(* CODESYS project PRO_JSON 1.0.20.0 Codesys SP17.library
   DocFormat: reStructuredText
   Company: Pro Electric
   DefaultNamespace: PRO_JSON
   Placeholder: PRO_JSON
   Author: TVM
   Description: Patched by Risele
   Version: 1.0.20.0
   Title: PRO JSON

Project tree, tasks and I/O mapping:
  libraries: Standard, 3.5.18.0 (System); StringUtils, 3.5.20.0 (System); SysMem, 3.5.17.0 (System); VisuDialogs, * (System)
  Data Types/
    data type ASCII
    data type JSONNAMEVALUE
    data type JSONVALUETYPE
    function block JSONVAR [ST]: FirstLevel, VarName, ValueType, Null, Number, Boolean, Integer, CharString, UInteger, Format, ApplicationLevel, LastIndex, ProgramLevel, AsUnicode, AsHexString, AsString, AsDWord, AsDateTime, Size, TestInit, Init, IsFirstVar, CreateNamesArray, FB_Init, GetArrayIndex
    data type JSONVARINFO
    data type JSONFORMAT
    data type ARRAY_INDEX
  Examples/
    data type EXAMPLEJSONSTRUCT
    data type EXAMPLEJSONSTRUCT_1
    program ExampleJSON_PRG [ST]
    function block EXAMPLE_FB [ST]
    program Test_ArrayOfStruct_PRG [ST]
    program Test_Array_PRG [ST]
    program Test_NestedStruct_PRG [ST]
    program Test_SingleVar_PRG [ST]
    program Test_Struct_PRG [ST]
    data type ARRAYOFSTRUCT
    data type JSONSTRUCT
    data type JSONSTRUCT_1
  Functions/
    function CLEANSTRING [ST]
    function ISBOOLEAN [ST]
    function ISNUMBER [ST]
    function REAL_TO_STRING_X [ST]
    function SPLIT_VARNAME [ST]
    function ISINTEGER [ST]
    function JSONVALUE_TO_STRING [ST]
    function STRING_TO_JSONVALUE [ST]
    function MATCH_NAMES [ST]
    function HEXSTR_TO_UDINT [ST]
    function ISHEX [ST]
    function UDINT_TO_HEXSTR [ST]
    function FORMAT_JSON [ST]
    function HEX4_TO_UINT [ST]
    function UINT_TO_HEX4 [ST]
    function VALUETYPE_FROM_STRING [ST]
    function ISNULL [ST]
    function DWORD_TO_HEXSTR [ST]
    function IEC_TO_JSON [ST]
    function JSON_TO_IEC [ST]
    function DWORD_TO_UNICODE [ST]
    function ARRAY_INDEXES_EQUAL [ST]
    function ARRAY_INDEXES_LESS [ST]
    function CLEAR_ARRAY_INDEX_VECTOR [ST]
  global variables GPL_JSON
  program Notes [ST]
  Visualizations/
    visualisation JSON_TO_STRUCT_VISU
    visualisation STRUCT_TO_JSON_VISU
    visualisation JSONVARS_TABLE_VISU
    visualisation JSONVAR_TABLE_VISU
    text list ValueType_Textlist
  text list GlobalTextList
  Function Blocks/
    function block JSON_TO_STRUCT [ST]: ClearAll, Value, FindValueStartPosition, GetValueAsString, FindValueStopPosition, ErrorHandler, ClearNameValue, CheckApplicationName, CheckMaxVars, CheckPointers, MatchAllLevels, CloseObject, OpenArray, Comma, CloseArray, OpenObject, Name
    function block STRUCT_TO_JSON [ST]: FindMaxLevel, CreateArray, CreateObject, CreateValue, CreateName, HasNonNullDescendant, PrependComma, Initialize, InitJsonVars, CheckMaxVars, CheckApplicationName, CheckPointers, FindMatchingClose, CloseArray, CloseObject, ClearString
*)

// Data Types/ASCII
///
///| Author: Tim Van Meppelen, Pro Electric Inc.
///| timv@proelectric.com
///| Date: Nov 2, 2018
///| enumeration of all ascii characters
TYPE ASCII :
(
	NULL := 0,
	SOH := 1,
	STX := 2,
	ETX := 3,
	EOT := 4,
	ENQ := 5,
	ACK := 6,
	BEL := 7,
	BS := 8,
	HT := 9,
	LF := 10,
	VT := 11,
	FF := 12,
	CR := 13,
	SO := 14,
	SI := 15,
	DLE := 16,
	DC1 := 17,
	DC2 := 18,
	DC3 := 19,
	DC4 := 20,
	NAK := 21,
	SYN := 22,
	ETB := 23,
	CAN := 24,
	EM := 25,
	SUB_ := 26,
	ESC := 27,
	FS := 28,
	GS := 29,
	RS := 30,
	US := 31,
	SPACE := 32,
	BANG := 33,
	DOUBLE_QUOTE := 34,
	HASH := 35,
	DOLLAR := 36,
	PERCENT := 37,
	AMPERSAND := 38,
	SINGLE_QUOTE := 39,
	OPEN_PAREN := 40,
	CLOSE_PAREN := 41,
	STAR := 42,
	PLUS := 43,
	COMMA := 44,
	MINUS := 45,
	DOT := 46,
	SLASH := 47,
	_0 := 48,
	_1 := 49,
	_2 := 50,
	_3 := 51,
	_4 := 52,
	_5 := 53,
	_6 := 54,
	_7 := 55,
	_8 := 56,
	_9 := 57,
	COLON := 58,
	SEMICOLON := 59,
	LESS_THAN := 60,
	EQUALS := 61,
	GREATER_THAN := 62,
	QUESTION := 63,
	AT_SIGN := 64,
	_A := 65,
	_B := 66,
	_C := 67,
	_D := 68,
	_E := 69,
	_F := 70,
	_G := 71,
	_H := 72,
	_I := 73,
	_J := 74,
	_K := 75,
	_L := 76,
	_M := 77,
	_N := 78,
	_O := 79,
	_P := 80,
	_Q := 81,
	_R := 82,
	_S := 83,
	_T := 84,
	_U := 85,
	_V := 86,
	_W := 87,
	_X := 88,
	_Y := 89,
	_Z := 90,
	OPEN_BRACKET := 91,
	BACKSLASH := 92,
	CLOSE_BRACKET := 93,
	CARET := 94,
	UNDERSCORE := 95,
	BACKQUOTE := 96,
	_a_ := 97,
	_b_ := 98,
	_c_ := 99,
	_d_ := 100,
	_e_ := 101,
	_f_ := 102,
	_g_ := 103,
	_h_ := 104,
	_i_ := 105,
	_j_ := 106,
	_k_ := 107,
	_l_ := 108,
	_m_ := 109,
	_n_ := 110,
	_o_ := 111,
	_p_ := 112,
	_q_ := 113,
	_r_ := 114,
	_s_ := 115,
	_t_ := 116,
	_u_ := 117,
	_v_ := 118,
	_w_ := 119,
	_x_ := 120,
	_y_ := 121,
	_z_ := 122,
	OPEN_BRACE := 123,
	PIPE := 124,
	CLOSE_BRACE := 125,
	TILDE := 126,
	DEL := 127
) BYTE;
END_TYPE

// Data Types/JSONNAMEVALUE
///
///| Author: Tim Van Meppelen, Pro Electric Inc.
///| timv@proelectric.com
///| Date: Nov 2, 2018
///| name : value pair
TYPE JSONNAMEVALUE :
STRUCT
	///name of the object at this level
	Name: STRING(GPL_JSON.MAX_NAME_SIZE);
	///value of the object at this level
	Value: STRING(GPL_JSON.MAX_VALUE_SIZE);
	///array index of the object at this level
	ArrayIndex: ARRAY_INDEX := ARRAY_INDEX.Invalid;
	IsArray: BOOL;
	ArrayDimCount: UINT := 0;
	ArrayIndexes: ARRAY[1..GPL_JSON.MAX_ARRAY_DIMENSIONS] OF INT;
END_STRUCT
END_TYPE

// Data Types/JSONVALUETYPE
///
///| Author: Tim Van Meppelen, Pro Electric Inc.
///| timv@proelectric.com
///| Date: Nov 2, 2018
///| enumeration of all json types
///| NOTE: JSON standard is somewhat ambiguous with number types, so integer and floating point numbers are separate types in this library
TYPE JSONVALUETYPE :
(
	///local var is type STRING
	json_string,
	///local var is REAL
	json_number,
	///local var is DINT
	json_integer,
	///locar var is UDINT	(new type by Fabrizio Morlino)
	json_uinteger,
	///local var is BOOL
	json_boolean,
	///local var is type null
	json_null,
	///object is an array
	json_array,
	///object is another object (nested objects)
	json_object
);
END_TYPE

// Data Types/JSONVARINFO
///
///| Author: Tim Van Meppelen, Pro Electric Inc.
///| timv@proelectric.com
///| Date: Nov 2, 2018
///| variable info structure, used with JSONVAR
TYPE JSONVARINFO :
STRUCT
	///name of this variable or object
	Name: STRING(GPL_JSON.MAX_NAME_SIZE);
	///first variable of a new object
	NewObject: BOOL;
	///variable in an object
	InObject: BOOL;
	///last variable of an object
	EndObject: BOOL;
	///array index of the object at this level	
	ArrayIndex: ARRAY_INDEX := ARRAY_INDEX.Invalid;
	///first variable of a new array
	NewArray: BOOL;
	///variable in an array
	InArray: BOOL;
	///last variable of an array
	EndArray: BOOL;
	/// 0 = not in array, 1..MAX_ARRAY_DIMENSIONS otherwise
	ArrayDimCount: UINT := 0;
	/// full multidim index vector
	ArrayIndexes: ARRAY[1..GPL_JSON.MAX_ARRAY_DIMENSIONS] OF INT;
END_STRUCT
END_TYPE

// Examples/EXAMPLEJSONSTRUCT
///
///| Author: Tim Van Meppelen, Pro Electric Inc.
///| timv@proelectric.com
///| Date: Jan 31, 2020
///| example of a struct of json variables
TYPE EXAMPLEJSONSTRUCT :
STRUCT
	var1: JSONVAR;
	var2: JSONVAR;
	var3: JSONVAR;
	obj: EXAMPLEJSONSTRUCT_1;
	arrayobj: ARRAY[1..3] OF JSONVAR;
END_STRUCT
END_TYPE

// Examples/EXAMPLEJSONSTRUCT_1
///
///| Author: Tim Van Meppelen, Pro Electric Inc.
///| timv@proelectric.com
///| Date: Jan 31, 2020
///| example of a struct of json variables
TYPE EXAMPLEJSONSTRUCT_1 :
STRUCT
	var4: JSONVAR;
	var5: JSONVAR;
	var6: JSONVAR;
	var7: ARRAY[1..3] OF JSONVAR;
END_STRUCT
END_TYPE

// Examples/ARRAYOFSTRUCT
TYPE ARRAYOFSTRUCT :
STRUCT
	arr: ARRAY[1..4] OF JSONSTRUCT;
END_STRUCT
END_TYPE

// Examples/JSONSTRUCT
TYPE JSONSTRUCT :
STRUCT
	obj1: JSONVAR;
	_obj2: JSONVAR;
	obj3: JSONVAR;
END_STRUCT
END_TYPE

// Examples/JSONSTRUCT_1
TYPE JSONSTRUCT_1 :
STRUCT
	obj1: JSONVAR;
	obj2: JSONVAR;
	obj3: JSONVAR;
	nest: JSONSTRUCT;
END_STRUCT
END_TYPE

// Data Types/JSONFORMAT
{attribute 'qualified_only' := ''}
{attribute 'strict' := ''}
TYPE JSONFORMAT :
(
	Undefined,
	Hex,
	Unicode,
	Decimal,
	Binary,
	DateTime
);
END_TYPE

// Data Types/ARRAY_INDEX
TYPE ARRAY_INDEX :
(
	Invalid:= -999
);
END_TYPE

// GPL_JSON
///
///| Author: Tim Van Meppelen, Pro Electric Inc.
///| timv@proelectric.com
///| Date: June 26, 2018
///| Parameter list that contains limits on size of strings, arrays, etc.  Most of these variables are simply
///| to limit memory usage, so they can be increased or decreased to suit the local application and controller
{attribute 'parameterlist' := ''}
{attribute 'qualified_only' := ''}
VAR_GLOBAL CONSTANT
	///maximum number of nested object levels
	MAX_LEVELS: UINT := 10;
	///max string length of JSON name
	MAX_NAME_SIZE: UINT := 20;
	///max value size in bytes (all values are this size in memory)
	MAX_VALUE_SIZE: UINT := 20;
	///maximum length of full variable name with path
	MAX_VAR_NAME: UINT := 150;
	///maximum number of variables in the local structure
	MAX_VARS: UINT := 1500;
	///maximum time for a single scan of the JSON_TO_STRUCT function block
	MAX_EXECUTION_TIME: TIME := TIME#50ms;
	///maximum allowable size of JSON string
	MAX_JSON_STRING: UINT := 20000;
	///formatting string for new line
	NEWLINE: STRING(2) := '$R$N';
	///formatting string for indentation
	INDENT: STRING(5) := '    ';
	///ignore first character in variable names
	IGNORE_LEADING_CHAR: STRING(1) := '_';
	///must match the name of your application
	APPLICATION_NAME: STRING(GPL_JSON.MAX_NAME_SIZE) := 'Application';
	///maximum array dimensions for multi-dimensional arrays
	MAX_ARRAY_DIMENSIONS: UINT := 3;
	(*
	When source array dimensions exceed GPL_JSON.MAX_ARRAY_DIMENSIONS:
	TRUE  : flatten overflow dimensions into the last kept dimension.
	FALSE : do not flatten overflow into the last kept dimension (overflow follows non-flatten branch behavior).
	
	Note: values are preserved; only array nesting/grouping (JSON shape) changes.
	*)
	FLATTEN_OVERFLOW_INTO_LAST_DIM : BOOL := FALSE;
	///support JSON5 hex strings
	JSON5: BOOL := TRUE;
	///  Suppress the codesys variable name appearing as root object. Could be overriden at parser params
	ROOTLESS: BOOL := FALSE;
END_VAR

// Notes
(*
| Author: Tim Van Meppelen, Pro Electric Inc.
| timv@proelectric.com
| Date: Nov 2, 2018
| 
| Tested with 200mS cyclic task, GPL_JSON.MAX_EXECUTION_TIME=50mS
| Depending on the application and speed of the controller, these values could be changed. 
| Be aware of how much cycle time is being taken when using multiple function blocks.
| Each function block will limit its time to GPL_JSON.MAX_EXECUTION_TIME, but multiple function blocks 
| could take up more than that.  This is on the list of things that could be improved. 
| 
| JSONVAR
| FB_Init will fill in information about the variable name and structure in VarNameArray
| variable type and size are automatically determined when a value is set, either:
| 	-with the set accessor of the AsString Property, which will make a guess at the type, based on the value
| 	-with any of the set accessors of the CharString, Boolean, Integer, Number, or Null properties
| variable name is set automatically in FB_Init
| 	-variable name is the JSON name
| 	-JSON allows some object names that are not valid variable names in IEC61131, for example "type", 
| 	"3h", etc.  Workaround is to put an underscore at the beginning of the variable name.  This will
| 	match in JSON_TO_STRUCT, and STRUCT_TO_JSON will create a name without the leading underscore
| 	
| JSON_TO_STRUCT
| convert a JSON string into a local structure of JSONVAR
| Long strings can take several seconds--for example, I have tested with a string of 20kB length, and the 
| parse time is about 4 seconds.  Ensuring that the local variable structure is designed to be as close as 
| possible to the expected order of variables in the JSON string will decrease parsing time, the search loop 
| always starts with the next local variable and loops around until a match is found.
| 
| STRUCT_TO_JSON
| convert a local structure of JSONVAR to a JSON string
| .Format input will create indenting and new lines, useful for writing to a file TO DO: not tested yet
| 
| GPL_JSON
| Parameter list that contains limits on size of strings, arrays, etc.  Most of these variables are simply
| to limit memory usage, so they can be increased or decreased to suit the local application and controller
*)
PROGRAM Notes

END_PROGRAM

// Data Types/JSONVAR
///
///| Author: Tim Van Meppelen, Pro Electric Inc.
///| timv@proelectric.com
///| Date: Nov 2, 2018
///| local JSON variables
///| 
///| for use with JSON_TO_STRUCT, STRUCT_TO_JSON
///| variable type and size are automatically determined when a value is set, either:
///| 
///| - with the set accessor of the AsString Property, which will make a guess at the type, based on the value
///| - with any of the set accessors of the CharString, Boolean, Integer, Number, or Null properties
///| 
///| variable name is set automatically in FB_Init:
///| 
///| - variable name is the JSON name
///| - JSON allows some object names that are not valid variable names in IEC61131, for example "type", "3h", etc.  
///| Workaround is to put a character (default: underscore) at the beginning of the variable name.  This will match in JSON_TO_STRUCT, 
///| and STRUCT_TO_JSON will create a name without the leading underscore.  Character can be changed in GPL_JSON.IGNORE_LEADING_CHAR
///
///{attribute 'hide_all_locals'}
{attribute 'pack_mode' := '4'}
{attribute 'reflection' := ''}
{attribute 'symbol' := 'none'}
FUNCTION_BLOCK JSONVAR
VAR_INPUT
	///variable info as an array. [1] is variable this var, [2..x] are higher levels	
	JSONVarInfo: ARRAY[1..GPL_JSON.MAX_LEVELS] OF JSONVARINFO;
END_VAR
VAR
	///JSON name uses the variable name
	{attribute 'instance-path' := ''}
	{attribute 'noinit'}
	_VarNameFull: STRING(GPL_JSON.MAX_VAR_NAME);
	///type of variable contained in the value field, also implicity defines size of local var
	_ValueType: JSONVALUETYPE := JSONVALUETYPE.json_null;
	///value stored internally as an array of bytes
	_InternalValue: ARRAY[1..(GPL_JSON.MAX_VALUE_SIZE + 1)] OF BYTE;
	///size of internal value in bytes, automatically determined when any of the type properties are set
	_Size: UINT;
	///array position which points to the application
	_ApplicationLevel: INT;
	///flag that the first element was initialized in STRUCT_TO_JSON.Init method
	_InitDone: BOOL;
	///for use by STRUCT_TO_JSON, index of last element in this structure or array
	_LastIndex: UDINT;
	///format information for composing
	_Format: JSONFORMAT;
END_VAR
VAR_OUTPUT
	///this output is updated every time AsString property is set, for use with external HMI through symbol configuration
	{attribute 'symbol' := 'read'}
	HMIVarAsString: STRING(GPL_JSON.MAX_VALUE_SIZE);
END_VAR
VAR_STAT
	///previous JSONVAR
	PrevVar: REFERENCE TO JSONVAR;
END_VAR

(* Notes on variable attributes

The only thing we have to work with is _VarNameFull.  Some examples:

ARRAY[1..2] OF JSONVAR
Device.Application.Program.TestJSONStruct.var1
Device.Application.Program.TestJSONStruct.var2
Device.Application.Program.TestJSONStruct.var3
Device.Application.Program.TestJSONStruct.var4
{"var1": 1, "var2": true, "var3": "hello", "var4": 4.342}

ARRAY[1..2] OF JSONVAR
Device.Application.Program.TestJSONStruct.Arr1[1]
Device.Application.Program.TestJSONStruct.Arr1[2]
Device.Application.Program.TestJSONStruct.Arr2[1]
Device.Application.Program.TestJSONStruct.Arr2[2]
{"Arr1"[1,2], "Arr2"[3,4]}

ARRAY[1..2] OF STRUCT <-which contains 2 JSONVAR
Device.Application.Program.TestJSONStruct.Arr1[1].var1
Device.Application.Program.TestJSONStruct.Arr1[1].var2
Device.Application.Program.TestJSONStruct.Arr1[2].var1
Device.Application.Program.TestJSONStruct.Arr1[2].var2
{"Arr1"[{"var1": 1, "var2": 2}, {"var1": 1, "var2": 2}]}

nested objects/structs
Device.Application.Program.TestJSONStruct.outer.inner.var1
Device.Application.Program.TestJSONStruct.outer.inner.var2
Device.Application.Program.TestJSONStruct.outer.inner.var3
Device.Application.Program.TestJSONStruct.outer.var1
Device.Application.Program.TestJSONStruct.var1
{"outer":{"inner":{"var1":1,"var2":2,"var3":3},"var1":1},"var1":1}

Example:  'Device.Application.Program.TestJSONStruct.Arr1[1].objname'
[1] objname
[2] Arr1 (with array index of 1)
[3] TestJSONStruct
[4] Program
[5] Application
-Application name must match GPL_JSON.APPLICATION_NAME, and is only used to establish a reference point
-one level below Application will always be a Program
-we don't care about anything above the Program level
-after that, levels could be any combination of function blocks and structures up to GPL_JSON.MAX_LEVELS
-index [1] is always the JSONVAR itself
-offset is used to determine how far nesting has shifted up(+) or down(-)

*)

{attribute 'monitoring' := 'call'}
PROPERTY FirstLevel : INT
GET
FirstLevel:= _ApplicationLevel - 2;
END_GET
END_PROPERTY

{attribute 'monitoring' := 'call'}
PROPERTY VarName : STRING(GPL_JSON.MAX_VAR_NAME)
SET
VAR
	Levels: UINT;
	i: INT;
END_VAR
Levels:= SPLIT_VARNAME(VarNameArray:= JSONVarInfo, StringIn:= VarName);

FOR i:= UINT_TO_INT(Levels) TO 1 BY -1 DO 
//recreate the var name string
	IF (i = UINT_TO_INT(Levels)) THEN
		_VarNameFull:= CONCAT(JSONVarInfo[i].Name,'.');
	ELSIF (i = 1) THEN
		_VarNameFull:= CONCAT(_VarNameFull, JSONVarInfo[i].Name);
	ELSE
		_VarNameFull:= CONCAT(_VarNameFull, JSONVarInfo[i].Name);
		_VarNameFull:= CONCAT(_VarNameFull, '.');
	END_IF
END_FOR
END_SET
GET
VarName:= _VarNameFull;
END_GET
END_PROPERTY

{attribute 'monitoring' := 'call'}
PROPERTY ValueType : JSONVALUETYPE
SET
_ValueType:= ValueType;
END_SET
GET
ValueType:= _ValueType;
END_GET
END_PROPERTY

{attribute 'monitoring' := 'call'}
PROPERTY Null : STRING(4)
GET
Null:= 'null';
END_GET
SET
_ValueType:= JSONVALUETYPE.json_null;
_Size:= 4;
END_SET
END_PROPERTY

{attribute 'monitoring' := 'call'}
PROPERTY Number : REAL
SET
_ValueType:= JSONVALUETYPE.json_number;
_Size:= 4;

//clear memory
SysMemSet(
	pDest:= ADR(_InternalValue), 
	udiValue:= 0, 
	udiCount:= SIZEOF(_InternalValue)
);

//put data into internal value
SysMemCpy(
	pDest:= ADR(_InternalValue), 
	pSrc:= ADR(Number), 
	udiCount:= _Size
);
END_SET
GET
VAR
	tempDINT: DINT;
	tempREAL: REAL;
END_VAR
CASE _ValueType OF
JSONVALUETYPE.json_integer:
//internal value was stored as integer, convert to floating point
	SysMemCpy(
		pDest:= ADR(tempDINT), 
		pSrc:= ADR(_InternalValue), 
		udiCount:= 4
	);
	Number:= DINT_TO_REAL(tempDINT);	
	
JSONVALUETYPE.json_number:
//internal value was stored as floating point, get value
	SysMemCpy(
		pDest:= ADR(tempREAL), 
		pSrc:= ADR(_InternalValue), 
		udiCount:= 4
	);
	Number:= tempREAL;	
END_CASE
END_GET
END_PROPERTY

{attribute 'monitoring' := 'call'}
PROPERTY Boolean : BOOL
SET
_ValueType:= JSONVALUETYPE.json_boolean;
_Size:= 1;

//clear memory
SysMemSet(
	pDest:= ADR(_InternalValue), 
	udiValue:= 0, 
	udiCount:= SIZEOF(_InternalValue)
);

//put data into internal value
SysMemCpy(
	pDest:= ADR(_InternalValue), 
	pSrc:= ADR(Boolean), 
	udiCount:= _Size
);
END_SET
GET
Boolean:= BYTE_TO_BOOL(_InternalValue[1]);
END_GET
END_PROPERTY

{attribute 'monitoring' := 'call'}
PROPERTY Integer : DINT
SET
VAR
	TempVar: DINT;
END_VAR
_ValueType:= JSONVALUETYPE.json_integer;
_Size:= 4;

//clear memory
SysMemSet(
	pDest:= ADR(_InternalValue), 
	udiValue:= 0, 
	udiCount:= SIZEOF(_InternalValue)
);

TempVar:= Integer;

//put data into internal value
SysMemCpy(
	pDest:= ADR(_InternalValue), 
	pSrc:= ADR(TempVar), 
	udiCount:= _Size
);
END_SET
GET
VAR
	tempDINT: DINT;
	tempREAL: REAL;
END_VAR
CASE _ValueType OF
JSONVALUETYPE.json_number:
//internal value was stored as floating point, convert to integer
	SysMemCpy(
		pDest:= ADR(tempREAL), 
		pSrc:= ADR(_InternalValue), 
		udiCount:= 4
	);
	Integer:= REAL_TO_DINT(tempREAL);		
JSONVALUETYPE.json_integer:
//internal value was stored as integer, get the value
	SysMemCpy(
		pDest:= ADR(tempDINT), 
		pSrc:= ADR(_InternalValue), 
		udiCount:= 4
	);
	Integer:= tempDINT;
END_CASE
END_GET
END_PROPERTY

{attribute 'monitoring' := 'call'}
PROPERTY CharString : STRING(GPL_JSON.MAX_VALUE_SIZE)
SET
_ValueType:= JSONVALUETYPE.json_string;
_Size:= INT_TO_UINT(LEN(CharString));

//clear memory
SysMemSet(
	pDest:= ADR(_InternalValue), 
	udiValue:= 0, 
	udiCount:= SIZEOF(_InternalValue)
);

//put data into internal value
SysMemCpy(
	pDest:= ADR(_InternalValue), 
	pSrc:= ADR(CharString), 
	udiCount:= _Size+1
);
END_SET
GET
VAR
	TempVar: STRING(255);
END_VAR
SysMemCpy(
	pDest:= ADR(TempVar), 
	pSrc:= ADR(_InternalValue), 
	udiCount:= _Size+1
);
CharString:= TempVar;
END_GET
END_PROPERTY

{attribute 'monitoring' := 'call'}
PROPERTY UInteger : UDINT
SET
VAR
	TempVar: UDINT;
END_VAR
_ValueType:= JSONVALUETYPE.json_uinteger;
_Size:= 4;

//clear memory
SysMemSet(
	pDest:= ADR(_InternalValue), 
	udiValue:= 0, 
	udiCount:= SIZEOF(_InternalValue)
);

TempVar:= UInteger;

//put data into internal value
SysMemCpy(
	pDest:= ADR(_InternalValue), 
	pSrc:= ADR(TempVar), 
	udiCount:= _Size
);
END_SET
GET
VAR
	tempUDINT: UDINT;
	tempREAL: REAL;
END_VAR
CASE _ValueType OF
JSONVALUETYPE.json_number:
//internal value was stored as floating point, convert to uinteger
	SysMemCpy(
		pDest:= ADR(tempREAL), 
		pSrc:= ADR(_InternalValue), 
		udiCount:= 4
	);
	UInteger:= REAL_TO_UDINT(tempREAL);		
JSONVALUETYPE.json_uinteger:
//internal value was stored as integer, get the value
	SysMemCpy(
		pDest:= ADR(tempUDINT), 
		pSrc:= ADR(_InternalValue), 
		udiCount:= 4
	);
	UInteger:= tempUDINT;
END_CASE
END_GET
END_PROPERTY

{attribute 'monitoring' := 'call'}
PROPERTY Format : JSONFORMAT
SET
_Format:= Format;
END_SET
GET
Format:= _Format;
END_GET
END_PROPERTY

{attribute 'monitoring' := 'call'}
PROPERTY ApplicationLevel : INT
GET
ApplicationLevel:= _ApplicationLevel;
END_GET
END_PROPERTY

{attribute 'monitoring' := 'call'}
PROPERTY LastIndex : UDINT
SET
_LastIndex:= LastIndex;
END_SET
GET
LastIndex:= _LastIndex;
END_GET
END_PROPERTY

{attribute 'monitoring' := 'call'}
PROPERTY ProgramLevel : INT
GET
ProgramLevel:= _ApplicationLevel - 1;
END_GET
END_PROPERTY

{attribute 'monitoring' := 'call'}
PROPERTY AsUnicode : STRING(GPL_JSON.MAX_VALUE_SIZE)
SET
_ValueType:= JSONVALUETYPE.json_uinteger;
_Format:= JSONFORMAT.Hex;
UInteger:= HEXSTR_TO_UDINT(AsHexString);


HMIVarAsString:= AsString;
END_SET
GET
CASE _ValueType OF
JSONVALUETYPE.json_uinteger:
	AsUnicode := DWORD_TO_UNICODE(THIS^.UInteger);	
JSONVALUETYPE.json_number:
	AsUnicode := DWORD_TO_UNICODE(TO_DWORD(THIS^.Number));
JSONVALUETYPE.json_integer:
	AsUnicode := DWORD_TO_UNICODE(TO_DWORD(THIS^.Integer));
END_CASE
END_GET
END_PROPERTY

{attribute 'monitoring' := 'call'}
PROPERTY AsHexString : STRING(GPL_JSON.MAX_VALUE_SIZE)
SET
_ValueType:= JSONVALUETYPE.json_uinteger;
_Format:= JSONFORMAT.Hex;
UInteger:= HEXSTR_TO_UDINT(AsHexString);


HMIVarAsString:= AsString;
END_SET
GET
CASE _ValueType OF
JSONVALUETYPE.json_uinteger:
	AsHexString := DWORD_TO_HEXSTR(THIS^.UInteger);	
JSONVALUETYPE.json_number:
	AsHexString := DWORD_TO_HEXSTR(TO_DWORD(THIS^.Number));
JSONVALUETYPE.json_integer:
	AsHexString := DWORD_TO_HEXSTR(TO_DWORD(THIS^.Integer));
END_CASE
END_GET
END_PROPERTY

{attribute 'monitoring' := 'call'}
PROPERTY AsString : STRING(GPL_JSON.MAX_VALUE_SIZE)
SET
STRING_TO_JSONVALUE(
	In_String:= AsString,
	Out_JSON:= THIS
);

HMIVarAsString:= AsString;
END_SET
GET
AsString:= JSONVALUE_TO_STRING(THIS);
END_GET
END_PROPERTY

{attribute 'monitoring' := 'call'}
PROPERTY AsDWord : DWORD
GET
CASE _ValueType OF
JSONVALUETYPE.json_number:
	AsDWord:= REAL_TO_DWORD(THIS^.Number);
JSONVALUETYPE.json_integer:
	AsDWord:= DINT_TO_DWORD(THIS^.Integer);
JSONVALUETYPE.json_uinteger:
	AsDWord:= UDINT_TO_DWORD(THIS^.UInteger);
JSONVALUETYPE.json_string:
	AsDWord:= STRING_TO_DWORD(THIS^.CharString);
END_CASE
END_GET
SET
VAR
	TempReal: REAL;
	TempInt: DINT;
	TempUInt: UDINT;
	TempString: STRING;
END_VAR
CASE _ValueType OF
JSONVALUETYPE.json_number:
	TempReal:= DWORD_TO_REAL(AsDWord);
	THIS^.Number:= TempReal;
JSONVALUETYPE.json_integer:
	TempInt:= DWORD_TO_DINT(AsDWord);
	THIS^.Integer:= TempInt;	
JSONVALUETYPE.json_uinteger:
	TempUInt:= DWORD_TO_UDINT(AsDWord);
	THIS^.UInteger:= TempUInt;	
JSONVALUETYPE.json_string:
	TempString:= DWORD_TO_STRING(AsDWord);
	THIS^.CharString:= TempString;
END_CASE
END_SET
END_PROPERTY

{attribute 'monitoring' := 'call'}
PROPERTY AsDateTime : DT
GET
CASE _ValueType OF
JSONVALUETYPE.json_number:
	AsDateTime:= REAL_TO_DT(THIS^.Number);
JSONVALUETYPE.json_integer:
	AsDateTime:= DINT_TO_DT(THIS^.Integer);
JSONVALUETYPE.json_uinteger:
	AsDateTime:= UDINT_TO_DT(THIS^.UInteger);	
JSONVALUETYPE.json_string:
	AsDateTime:= STRING_TO_DT(THIS^.CharString);
END_CASE
END_GET
SET
VAR
	TempReal: REAL;
	TempInt: DINT;
	TempUInt: UDINT;
	TempString: STRING(255);
END_VAR
CASE _ValueType OF
JSONVALUETYPE.json_number:
	TempReal:= DT_TO_REAL(AsDateTime);
	THIS^.Number:= TempReal;
JSONVALUETYPE.json_integer:
	TempInt:= DT_TO_DINT(AsDateTime);
	THIS^.Integer:= TempInt;
JSONVALUETYPE.json_uinteger:
	TempUInt:= DT_TO_UDINT(AsDateTime);
	THIS^.UInteger:= TempUInt;		
JSONVALUETYPE.json_string:
	TempString:= DT_TO_STRING(AsDateTime);
	THIS^.CharString:= TempString;
END_CASE
_Format:= JSONFORMAT.DateTime;
END_SET
END_PROPERTY

{attribute 'monitoring' := 'call'}
PROPERTY Size : UINT
GET
Size:= _Size;
END_GET
END_PROPERTY

///
///| Author: Tim Van Meppelen, Pro Electric Inc.
///| timv@proelectric.com
///| Date: Nov 2, 2018
///| split the variable path into an array, and determine some object characteristics
///| example variable path: 'Device.Sim.Device.Application.TestJSON_PRG.TestJSONStruct.Arr1[1, 1].objname'
METHOD TestInit : BOOL
VAR
	NameStringPtr: POINTER TO ARRAY[1..GPL_JSON.MAX_VAR_NAME] OF BYTE;
	startarraystr: INT;
	endarraystr: INT;
	NumberOfLevels: INT;
	i: INT;
	offset: INT;
	varlevelindex: INT;
	prevvarlevelindex: INT;
	Count: INT;
	Indexes: ARRAY[1..GPL_JSON.MAX_ARRAY_DIMENSIONS] OF UINT;
END_VAR
//==================== GET VARIABLE NAMES INTO AN ARRAY ====================
//fill inthe JSONVarInfo array with the name and array indexes of each variable
CreateNamesArray();


//==================== JSON OBJECT CHARACTERISTICS ====================
(*VAR_STAT PrevVar is a reference to the last JSONVAR variable
that was worked on.  This would be the previous variable in a structure or array, but
could also be a variable contained in a completely different JSON structure.
Because it is not possible to reference the next variable in a structure (because
its FB_Init() method has not run yet), the characteristics of the last variable 
in a structure are set in the STRUCT_TO_JSON function block.*)

IF IsFirstVar() THEN
//this is the first variable of a structure of JSONVARs

	//==================== New object/in object ====================
	FOR varlevelindex:= 1 TO _ProgramLevel-1 DO
	//on the first variable, every new level above 1 creates a new object
		IF (varlevelindex > 1) THEN
			JSONVarInfo[varlevelindex].NewObject:= TRUE;
			JSONVarInfo[varlevelindex].InObject:= TRUE;
		END_IF
	
		//==================== New array ====================	
		IF (JSONVarInfo[varlevelindex].ArrayIndex <> ARRAY_INDEX.Invalid) THEN 
		//on the first variable, any array index creates a new array
			JSONVarInfo[varlevelindex].NewArray:= TRUE;
			JSONVarInfo[varlevelindex].InArray:= TRUE;
		END_IF
		
	END_FOR	
ELSE	
//not the first variable of a STRUCT
	offset:= _ApplicationLevel - PrevVar.ApplicationLevel;	//check if the variable names have shifted up or down
	FOR varlevelindex:= 1 TO _ProgramLevel-1 DO
		prevvarlevelindex:= varlevelindex - offset;	//tracks the equivalent level in the previous variable

		//==================== New array ====================
		IF (varlevelindex = 1) THEN
		//level 1
			IF (NOT PrevVar.JSONVarInfo[prevvarlevelindex].InArray) AND (JSONVarInfo[varlevelindex].ArrayIndex <> ARRAY_INDEX.Invalid) THEN
			//first array index on level 1 always indicates a new array	
				JSONVarInfo[varlevelindex].NewArray:= TRUE;
			END_IF
			
		ELSE
		//all other levels
			IF (NOT PrevVar.JSONVarInfo[prevvarlevelindex].InArray) AND 
			  (JSONVarInfo[varlevelindex].ArrayIndex <> ARRAY_INDEX.Invalid) AND
			  (PrevVar.JSONVarInfo[prevvarlevelindex].Name <> JSONVarInfo[varlevelindex].Name) THEN
			//first array index means the start of a new array
			//unless the array was already started in the previous var
			//as long as they have different names (adjacent array case) 	
				JSONVarInfo[varlevelindex].NewArray:= TRUE;
			END_IF
	
		END_IF

		//==================== End previous array ====================
		IF (offset < 0) AND (varlevelindex = 1) THEN
		//object levels have shifted down
			IF (PrevVar.JSONVarInfo[prevvarlevelindex].InArray) THEN
			//previous var was an array, and objects have shifted, therefore the array must be closed
				PrevVar.JSONVarInfo[prevvarlevelindex].EndArray:= TRUE;
			END_IF	
		ELSIF (offset = 0) THEN
		//object levels have not shifted
			IF JSONVarInfo[varlevelindex].NewArray AND PrevVar.JSONVarInfo[prevvarlevelindex].InArray THEN
			  //this var is a new array, close the previous one (adjacent arrays)
			  PrevVar.JSONVarInfo[prevvarlevelindex].EndArray:= TRUE;
			ELSIF ((JSONVarInfo[varlevelindex].ArrayIndex = ARRAY_INDEX.Invalid) AND PrevVar.JSONVarInfo[prevvarlevelindex].InArray) THEN
			//this var is not an array, but the previous one was, so close it
				PrevVar.JSONVarInfo[prevvarlevelindex].EndArray:= TRUE;
			END_IF
		END_IF

		//==================== In array ====================
		//TO DO:  these are probably not all necessary
		IF (JSONVarInfo[varlevelindex].ArrayIndex <> ARRAY_INDEX.Invalid) THEN
		//if there is an array index present
			JSONVarInfo[varlevelindex].InArray:= TRUE;
		ELSIF (varlevelindex > 1) AND PrevVar.JSONVarInfo[prevvarlevelindex].InArray THEN
		//previous var at same level is in array, this one must be as well
			JSONVarInfo[varlevelindex].InArray:= TRUE;
		ELSIF JSONVarInfo[varlevelindex].NewArray OR JSONVarInfo[varlevelindex].EndArray THEN
		//this var is the beginning or end of an array
			JSONVarInfo[varlevelindex].InArray:= TRUE;
		END_IF
		
		//==================== New object ====================
		IF (varlevelindex > 1) AND (offset > 0) THEN
		//object levels have shifted up, level 1 is always a variable, never an object
			IF PrevVar.JSONVarInfo[prevvarlevelindex].InObject THEN
			//previous var equivalent level was already an object
				JSONVarInfo[varlevelindex].InObject:= TRUE;
			ELSIF (varlevelindex = 2) THEN		//TO DO:  what about offset > 1?
			//we shifted, therefore a new object must have been created at level 2
				JSONVarInfo[varlevelindex].NewObject:= TRUE;
				JSONVarInfo[varlevelindex].InObject:= TRUE;				
			END_IF
		END_IF
		
		IF (varlevelindex > 1) 
			AND ((NOT JSONVarInfo[varlevelindex].NewArray) //not a new array
			AND (JSONVarInfo[varlevelindex].Name <> PrevVar.JSONVarInfo[prevvarlevelindex].Name) //names are different
			OR (JSONVarInfo[varlevelindex].ArrayIndex <> PrevVar.JSONVarInfo[prevvarlevelindex].ArrayIndex)) //array indexes are different
			THEN
			JSONVarInfo[varlevelindex].NewObject:= TRUE;	//new object at this level	
		END_IF
		
		//==================== End previous object ====================
		//IF (varlevelindex > 1) AND (offset <= 0)  AND
		IF (offset <= 0)  THEN
		//objects have shifted down, or no shift
		  IF PrevVar.JSONVarInfo[prevvarlevelindex].InObject AND (JSONVarInfo[varlevelindex].Name <> PrevVar.JSONVarInfo[prevvarlevelindex].Name) THEN
		  //previous var at same level is an object, and name doesn't match 
			PrevVar.JSONVarInfo[prevvarlevelindex].EndObject:= TRUE;	//close previous object	
			
			ELSIF PrevVar.JSONVarInfo[prevvarlevelindex].InArray AND (JSONVarInfo[varlevelindex].ArrayIndex <> PrevVar.JSONVarInfo[prevvarlevelindex].ArrayIndex) THEN
			//previous var at same level is an array, and array index doesn't match (for array of objects)
				PrevVar.JSONVarInfo[prevvarlevelindex].EndObject:= TRUE;	//close previous object	
			END_IF
		END_IF
		
		
		//TO DO:  EndObject TRUE by default, so the last var automatically closes
		//IF (offset <= 0)  AND
		////objects have shifted down, or no shift
		//  (JSONVarInfo[varlevelindex].Name = PrevVar.JSONVarInfo[prevvarlevelindex].Name) THEN
		//  //previous var name at same level matches
		//	PrevVar.JSONVarInfo[prevvarlevelindex].EndObject:= FALSE;	//don't close previous object	
		//ELSIF (varlevelindex > 1) THEN
		////no shift
		//	PrevVar.JSONVarInfo[prevvarlevelindex].EndObject:= FALSE;	//don't close previous object	
		//END_IF
		//
 		//IF (varlevelindex > 1) AND PrevVar.JSONVarInfo[prevvarlevelindex].NewObject OR PrevVar.JSONVarInfo[prevvarlevelindex].NewArray THEN
		////clear EndObject flags where not needed
		//	PrevVar.JSONVarInfo[prevvarlevelindex].EndObject:= FALSE;
		//END_IF
		
		//==================== In object ====================
		IF (varlevelindex > 1) AND PrevVar.JSONVarInfo[prevvarlevelindex].InObject THEN
		//previous var at same level is in object, this one must be as well
			JSONVarInfo[varlevelindex].InObject:= TRUE;
		ELSIF (JSONVarInfo[varlevelindex].NewObject OR JSONVarInfo[varlevelindex].EndObject) THEN
			JSONVarInfo[varlevelindex].InObject:= TRUE;
		END_IF
	END_FOR
END_IF

//FOR i:= _ProgramLevel TO TO_INT(GPL_JSON.MAX_LEVELS) DO
////EndObject is set to TRUE by default, clear all above program level
//	JSONVARInfo[i].EndObject:= FALSE;
//END_FOR

//save this variable reference as a reference for the next variable
PrevVar REF= THIS^;
END_METHOD

{attribute 'monitoring' := 'call'}
PROPERTY Init : BOOL
SET
_InitDone:= Init;
END_SET
GET
Init:= _InitDone;
END_GET
END_PROPERTY

///
///| Author: Tim Van Meppelen, Pro Electric Inc.
///| timv@proelectric.com
///| Date: June 16, 2025
///| is this the first var of a struct?
METHOD PRIVATE IsFirstVar : BOOL
//First variable of a structure
IF __ISVALIDREF(PrevVar) THEN
//there is a valid reference to a previous variable, check the previous object
	IF PrevVar.JSONVarInfo[PrevVar.ProgramLevel].Name <> JSONVarInfo[ProgramLevel].Name THEN
	//new program, must be a new variable
		IsFirstVar:= TRUE;
	ELSE
		IF PrevVar.JSONVarInfo[PrevVar.ProgramLevel-1].Name <> JSONVarInfo[ProgramLevel-1].Name THEN
		//new function block or main struct, must be a new variable
			IsFirstVar:= TRUE;
		END_IF
	END_IF

ELSE
//there is no valid reference to a previous variable, indicating that this is the first time FB_Init has run anywhere in the application
//therefore, this is the first variable of a new JSON object
	IsFirstVar:= TRUE;
END_IF
END_METHOD

///
///| Author: Tim Van Meppelen, Pro Electric Inc.
///| timv@proelectric.com
///| Date: Nov 2, 2018
///| split the variable path into an array
///| example variable path: 'Device.Sim.Device.Application.TestJSON_PRG.TestJSONStruct.Arr1[1, 1].objname'
///| called from FB_Init
METHOD PRIVATE CreateNamesArray
VAR
	NameStringPtr: POINTER TO ARRAY[1..GPL_JSON.MAX_VAR_NAME] OF BYTE;
	startarraystr: INT;
	endarraystr: INT;
	NumberOfLevels: INT;
	i: INT;
	offset: INT;
	varlevelindex: INT;
	prevvarlevelindex: INT;
	Count: INT;
	Indexes: ARRAY[1..GPL_JSON.MAX_ARRAY_DIMENSIONS] OF INT;
	j: UINT;
END_VAR
(*
General notes:
Example:  'Device.Sim.Device.Application.TestJSON_PRG.TestJSONStruct.Arr1[1, 1].objname'
[1] objname
[2] Arr1
[3] TestJSONStruct
[4] TestJSON_PRG
[5] Application
-we don't care about anything above the Application level.
-Application name must match GPL_JSON.APPLICATION_NAME
-one level below Application will always be a program
-after that, levels could be any combination of function blocks and structures up to GPL_JSON.MAX_LEVELS
-index [1] is always the name of the JSONVAR
*)

NameStringPtr:= ADR(_VarNameFull);
NumberOfLevels:= TO_INT(SPLIT_VARNAME(VarNameArray:= JSONVarInfo, StringIn:= _VarNameFull));

FOR i:= 1 TO NumberOfLevels DO
	IF (JSONVarInfo[i].Name = GPL_JSON.APPLICATION_NAME) THEN
		_ApplicationLevel:= i;
		EXIT;
	END_IF
END_FOR

FOR i:= 1 TO NumberOfLevels DO
	JSONVarInfo[i].ArrayDimCount := UINT#0;
	FOR j := 1 TO GPL_JSON.MAX_ARRAY_DIMENSIONS DO
		JSONVarInfo[i].ArrayIndexes[j] := ARRAY_INDEX.Invalid;
	END_FOR
	JSONVarInfo[i].ArrayIndex := ARRAY_INDEX.Invalid;

	startarraystr:= FIND(STR1:= JSONVarInfo[i].Name, STR2:= '[');
	endarraystr:= FIND(STR1:= JSONVarInfo[i].Name, STR2:= ']');

	IF (startarraystr <> 0) AND (endarraystr <> 0) THEN
		Indexes := GetArrayIndex(
			arrString := JSONVarInfo[i].Name,
			idxCount => Count
		);

		IF Count > 0 THEN
			JSONVarInfo[i].ArrayDimCount := TO_UINT(Count);
			FOR j := 1 TO TO_UINT(Count) DO
				JSONVarInfo[i].ArrayIndexes[j] := Indexes[j];
			END_FOR
			JSONVarInfo[i].ArrayIndex := JSONVarInfo[i].ArrayIndexes[JSONVarInfo[i].ArrayDimCount];
		END_IF

		JSONVarInfo[i].Name:= DELETE(
			STR:= JSONVarInfo[i].Name,
			LEN:= endarraystr-startarraystr+1,
			POS:= startarraystr
		);
	END_IF
END_FOR
END_METHOD

///
///| Author: Tim Van Meppelen, Pro Electric Inc.
///| timv@proelectric.com
///| Date: Nov 2, 2018
///| split the variable path into an array, and determine some object characteristics
///| example variable path: 'Device.Application.TestJSON_PRG.TestJSONStruct.Arr1[1].objname'
METHOD FB_Init : BOOL
VAR_INPUT
	/// TRUE: the retain variables are initialized (reset warm / reset cold)
	bInitRetains: BOOL;
	/// TRUE: the instance will be copied to the copy code afterward (online change)
	bInCopyCode: BOOL;
END_VAR
VAR
	NameStringPtr: POINTER TO ARRAY[1..GPL_JSON.MAX_VAR_NAME] OF BYTE;
	startarraystr: INT;
	endarraystr: INT;
	NumberOfLevels: INT;
	i: INT;
	offset: INT;
	varlevelindex: INT;
	prevvarlevelindex: INT;
	Count: INT;
	Indexes: ARRAY[1..GPL_JSON.MAX_ARRAY_DIMENSIONS] OF UINT;
END_VAR
//==================== GET VARIABLE NAMES INTO AN ARRAY ====================
//fill in the JSONVarInfo array with the name and array indexes of each variable
CreateNamesArray();


//==================== JSON OBJECT CHARACTERISTICS ====================
// VAR_STAT PrevVar is a reference to the last JSONVAR variable that was worked on.

IF IsFirstVar() THEN
//this is the first variable of a structure of JSONVARs

	//==================== New object/in object ====================
	FOR varlevelindex:= 1 TO ProgramLevel DO
	//on the first variable, every new level above 1 creates a new object
		IF (varlevelindex > 1) THEN
			JSONVarInfo[varlevelindex].NewObject:= TRUE;
			JSONVarInfo[varlevelindex].InObject:= TRUE;
		END_IF
	
		//==================== New array ====================
		IF (JSONVarInfo[varlevelindex].ArrayDimCount > 0)
		   OR (JSONVarInfo[varlevelindex].ArrayIndex <> ARRAY_INDEX.Invalid) THEN
		//on the first variable, any array index creates a new array
			JSONVarInfo[varlevelindex].NewArray:= TRUE;
			JSONVarInfo[varlevelindex].InArray:= TRUE;
		END_IF
		
	END_FOR	

ELSE	
//not the first variable of a STRUCT
	offset:= _ApplicationLevel - PrevVar.ApplicationLevel;	//check if the variable names have shifted up or down

	//==================== Close dropped levels on shift-down ====================
	IF (offset < 0) THEN
		FOR i := 1 TO -offset DO
			//close dropped arrays
			IF PrevVar.JSONVarInfo[i].InArray
			   OR (PrevVar.JSONVarInfo[i].ArrayDimCount > 0)
			   OR (PrevVar.JSONVarInfo[i].ArrayIndex <> ARRAY_INDEX.Invalid) THEN
				PrevVar.JSONVarInfo[i].EndArray := TRUE;
				PrevVar.JSONVarInfo[i].InArray := TRUE;
			END_IF

			//close dropped objects (level 1 is value level, not object level)
			IF (i > 1) AND (
				PrevVar.JSONVarInfo[i].InObject
				OR PrevVar.JSONVarInfo[i].NewObject
				OR PrevVar.JSONVarInfo[i].NewArray
			) THEN
				PrevVar.JSONVarInfo[i].EndObject := TRUE;
				PrevVar.JSONVarInfo[i].InObject := TRUE;
			END_IF
		END_FOR
	END_IF

	FOR varlevelindex:= 1 TO ProgramLevel DO
		prevvarlevelindex:= varlevelindex - offset;	//tracks equivalent level in previous variable

		//==================== New array ====================
		IF (NOT PrevVar.JSONVarInfo[prevvarlevelindex].InArray)
		   AND (
				(JSONVarInfo[varlevelindex].ArrayDimCount > 0)
				OR (JSONVarInfo[varlevelindex].ArrayIndex <> ARRAY_INDEX.Invalid)
		   ) THEN
		//start a new array if previous var is not an array and this one is
			JSONVarInfo[varlevelindex].NewArray:= TRUE;

		ELSIF
			(
				(
					(PrevVar.JSONVarInfo[prevvarlevelindex].ArrayDimCount > 0)
					OR (PrevVar.JSONVarInfo[prevvarlevelindex].ArrayIndex <> ARRAY_INDEX.Invalid)
				)
				AND
				(
					(JSONVarInfo[varlevelindex].ArrayDimCount > 0)
					OR (JSONVarInfo[varlevelindex].ArrayIndex <> ARRAY_INDEX.Invalid)
				)
				AND
				(
					NOT ARRAY_INDEXES_EQUAL(
						A := JSONVarInfo[varlevelindex].ArrayIndexes,
						ACount := JSONVarInfo[varlevelindex].ArrayDimCount,
						B := PrevVar.JSONVarInfo[prevvarlevelindex].ArrayIndexes,
						BCount := PrevVar.JSONVarInfo[prevvarlevelindex].ArrayDimCount
					)
				)
				AND
				ARRAY_INDEXES_LESS(
					A := JSONVarInfo[varlevelindex].ArrayIndexes,
					ACount := JSONVarInfo[varlevelindex].ArrayDimCount,
					B := PrevVar.JSONVarInfo[prevvarlevelindex].ArrayIndexes,
					BCount := PrevVar.JSONVarInfo[prevvarlevelindex].ArrayDimCount
				)
			) THEN
		//adjacent array rollover
			JSONVarInfo[varlevelindex].NewArray:= TRUE;
			PrevVar.JSONVarInfo[prevvarlevelindex].EndArray:= TRUE;
		END_IF

		//==================== End previous array ====================
		IF (offset < 0) AND (varlevelindex = 1) THEN
		//object levels have shifted down
			IF PrevVar.JSONVarInfo[prevvarlevelindex].InArray
			   OR (PrevVar.JSONVarInfo[prevvarlevelindex].ArrayDimCount > 0)
			   OR (PrevVar.JSONVarInfo[prevvarlevelindex].ArrayIndex <> ARRAY_INDEX.Invalid) THEN
				PrevVar.JSONVarInfo[prevvarlevelindex].EndArray:= TRUE;
			END_IF	

		ELSIF (offset = 0) THEN
		//object levels have not shifted
			IF JSONVarInfo[varlevelindex].NewArray
			   AND PrevVar.JSONVarInfo[prevvarlevelindex].InArray THEN
			//new array started, close previous one
				PrevVar.JSONVarInfo[prevvarlevelindex].EndArray:= TRUE;

			ELSIF
				(
					(JSONVarInfo[varlevelindex].ArrayDimCount = 0)
					AND (JSONVarInfo[varlevelindex].ArrayIndex = ARRAY_INDEX.Invalid)
				)
				AND PrevVar.JSONVarInfo[prevvarlevelindex].InArray THEN
			//current var not in array, previous was
				PrevVar.JSONVarInfo[prevvarlevelindex].EndArray:= TRUE;
			END_IF
		END_IF

		//==================== In array ====================
		IF (JSONVarInfo[varlevelindex].ArrayDimCount > 0)
		   OR (JSONVarInfo[varlevelindex].ArrayIndex <> ARRAY_INDEX.Invalid) THEN
		//if array indexes are present
			JSONVarInfo[varlevelindex].InArray:= TRUE;

		ELSIF (varlevelindex > 1) AND PrevVar.JSONVarInfo[prevvarlevelindex].InArray THEN
		//previous var at same level is in array
			JSONVarInfo[varlevelindex].InArray:= TRUE;

		ELSIF JSONVarInfo[varlevelindex].NewArray OR JSONVarInfo[varlevelindex].EndArray THEN
		//this var begins or ends an array
			JSONVarInfo[varlevelindex].InArray:= TRUE;
		END_IF
		
		//==================== New object ====================
		IF (varlevelindex > 1) AND (offset > 0) THEN
		//object levels shifted up
			IF PrevVar.JSONVarInfo[prevvarlevelindex].InObject THEN
				JSONVarInfo[varlevelindex].InObject:= TRUE;
			ELSIF (varlevelindex = 2) THEN
				JSONVarInfo[varlevelindex].NewObject:= TRUE;
				JSONVarInfo[varlevelindex].InObject:= TRUE;				
			END_IF
		END_IF
		
		IF (varlevelindex > 1)
			AND (
				(
					(NOT JSONVarInfo[varlevelindex].NewArray)
					AND (JSONVarInfo[varlevelindex].Name <> PrevVar.JSONVarInfo[prevvarlevelindex].Name)
				)
				OR
				(
					(JSONVarInfo[varlevelindex].ArrayDimCount <> PrevVar.JSONVarInfo[prevvarlevelindex].ArrayDimCount)
					OR
					(
						NOT ARRAY_INDEXES_EQUAL(
							A := JSONVarInfo[varlevelindex].ArrayIndexes,
							ACount := JSONVarInfo[varlevelindex].ArrayDimCount,
							B := PrevVar.JSONVarInfo[prevvarlevelindex].ArrayIndexes,
							BCount := PrevVar.JSONVarInfo[prevvarlevelindex].ArrayDimCount
						)
					)
				)
			)
		THEN
			JSONVarInfo[varlevelindex].NewObject:= TRUE;
		END_IF
		
		//==================== End previous object ====================
		IF (offset <= 0) THEN
		//objects shifted down or no shift
			IF PrevVar.JSONVarInfo[prevvarlevelindex].InObject
			   AND (JSONVarInfo[varlevelindex].Name <> PrevVar.JSONVarInfo[prevvarlevelindex].Name) THEN
				PrevVar.JSONVarInfo[prevvarlevelindex].EndObject:= TRUE;

			ELSIF (varlevelindex > 1)
			  AND PrevVar.JSONVarInfo[prevvarlevelindex].InArray
			  AND (
					(JSONVarInfo[varlevelindex].ArrayDimCount <> PrevVar.JSONVarInfo[prevvarlevelindex].ArrayDimCount)
					OR
					(
						NOT ARRAY_INDEXES_EQUAL(
							A := JSONVarInfo[varlevelindex].ArrayIndexes,
							ACount := JSONVarInfo[varlevelindex].ArrayDimCount,
							B := PrevVar.JSONVarInfo[prevvarlevelindex].ArrayIndexes,
							BCount := PrevVar.JSONVarInfo[prevvarlevelindex].ArrayDimCount
						)
					)
				  ) THEN
				PrevVar.JSONVarInfo[prevvarlevelindex].EndObject:= TRUE;
			END_IF
		END_IF
		
		//==================== In object ====================
		IF (varlevelindex > 1) AND PrevVar.JSONVarInfo[prevvarlevelindex].InObject THEN
			JSONVarInfo[varlevelindex].InObject:= TRUE;
		ELSIF (JSONVarInfo[varlevelindex].NewObject OR JSONVarInfo[varlevelindex].EndObject) THEN
			JSONVarInfo[varlevelindex].InObject:= TRUE;
		END_IF

	END_FOR
END_IF

//save this variable reference as a reference for the next variable
PrevVar REF= THIS^;
END_METHOD

METHOD PRIVATE GetArrayIndex : ARRAY[1..GPL_JSON.MAX_ARRAY_DIMENSIONS] OF INT
VAR_INPUT
	/// e.g. "Arr1[1,2,3]"
	arrString: STRING(GPL_JSON.MAX_VAR_NAME);
END_VAR
VAR_OUTPUT
	/// count of parsed indices	
	idxCount: INT := 0;
END_VAR
VAR
	posStart: INT := 0;
	posEnd: INT := 0;
	content: STRING(GPL_JSON.MAX_VAR_NAME);
	token: STRING(GPL_JSON.MAX_VAR_NAME);
	ch: STRING(1);
	i: INT;
END_VAR

idxCount := 0;
FOR i := 1 TO TO_INT(GPL_JSON.MAX_ARRAY_DIMENSIONS) DO
    GetArrayIndex[i] := ARRAY_INDEX.Invalid;
END_FOR

FOR i := 1 TO LEN(arrString) DO
    IF MID(STR := arrString, LEN := 1, POS := i) = '[' THEN
        posStart := i;
        EXIT;
    END_IF
END_FOR

IF posStart > 0 THEN
    FOR i := posStart + 1 TO LEN(arrString) DO
        IF MID(STR := arrString, LEN := 1, POS := i) = ']' THEN
            posEnd := i;
            EXIT;
        END_IF
    END_FOR
END_IF

IF (posStart = 0) OR (posEnd <= posStart) THEN
    RETURN;
END_IF

content := MID(STR := arrString, LEN := posEnd - posStart - 1, POS := posStart + 1);
token := '';

FOR i := 1 TO LEN(content) DO
    ch := MID(STR := content, LEN := 1, POS := i);

    IF (ch = ' ') OR (ch = '\t') THEN
        CONTINUE;
    END_IF

    IF ((ch >= '0') AND (ch <= '9')) OR (ch = '-') THEN
        token := CONCAT(token, ch);
    END_IF

    IF (ch = ',') OR (i = LEN(content)) THEN
        IF token <> '' THEN
            IF idxCount < TO_INT(GPL_JSON.MAX_ARRAY_DIMENSIONS) THEN
                idxCount := idxCount + 1;
                GetArrayIndex[idxCount] := STRING_TO_INT(token);
            ELSIF NOT GPL_JSON.FLATTEN_OVERFLOW_INTO_LAST_DIM  THEN
                IF GPL_JSON.MAX_ARRAY_DIMENSIONS > 0 THEN
                    GetArrayIndex[GPL_JSON.MAX_ARRAY_DIMENSIONS] := STRING_TO_INT(token);
                    idxCount := TO_INT(GPL_JSON.MAX_ARRAY_DIMENSIONS);
                END_IF
            END_IF
            token := '';
        END_IF
    END_IF
END_FOR
END_METHOD

END_FUNCTION_BLOCK

// Function Blocks/JSON_TO_STRUCT
///
///| Author: Tim Van Meppelen, Pro Electric Inc.
///| timv@proelectric.com
///| Date: Nov 2, 2018
///| Last Modified: Oct 31, 2023
///| parse JSON string and place the values in a matching local structure of type JSONVAR
FUNCTION_BLOCK JSON_TO_STRUCT
VAR_INPUT
	///rising edge triggers parse of JSON string
	Execute: BOOL;
	///rising edge stops parsing of JSON string
	Abort: BOOL;
	///pointer to JSON string
	JSONString: POINTER TO ARRAY[1..GPL_JSON.MAX_JSON_STRING] OF ASCII;
	///size of string in bytes
	JSONStringSize: UDINT;
	///pointer to local structure made up of type JSONVAR
	JSONVars: POINTER TO ARRAY[1..GPL_JSON.MAX_VARS] OF JSONVAR;
	///number of variables in the local structure or array
	NumberOfVars: UDINT;
END_VAR
VAR_OUTPUT
	///busy parsing a string
	Busy: BOOL;
	///successfully parsed the whole string with no errors
	Done: BOOL;
	///parsing aborted by Abort input
	Aborted: BOOL;
	///unexpected character detected, string not completely parsed
	Error: BOOL;
	///character position where the unexpected character was found
	ErrorPosition: UDINT;
	///time it took to parse the string
	ParseTime: TIME;
	///error information
	ErrorMsg: STRING;
END_VAR
VAR
	///current position in the string
	bufferposition: UDINT;
	///name:value pair currently being worked on 
	NameValue: ARRAY[1..GPL_JSON.MAX_LEVELS] OF JSONNAMEVALUE;
	///number of nested objects
	obj_level: UINT;
	///valid name was found
	nameok: BOOL;
	///valid value found
	valueok: BOOL;
	///found a matching local var by name
	namesmatch: BOOL;
	jsonvarindex: UDINT;
	levelindex: UINT;
	nameindex: UINT;
	///time the current loop started
	thisloopstarttime: TIME;
	///time parsing started
	starttime: TIME;
	Execute_TRIG: R_TRIG;
	Abort_TRIG: R_TRIG;
	findloop: UDINT;
	parse: BOOL;
	ArrayOverflowDepth: ARRAY[1..GPL_JSON.MAX_LEVELS] OF UINT;
	ArrayTrackedDepth: ARRAY[1..GPL_JSON.MAX_LEVELS] OF UINT;
END_VAR

//input checks
IF NOT CheckPointers() THEN RETURN; END_IF;
IF NOT CheckMaxVars() THEN RETURN; END_IF;
IF NOT CheckApplicationName() THEN RETURN; END_IF;

thisloopstarttime:= TIME();	//store the time of the beginning of this loop	

Execute_TRIG(CLK:= Execute);
Abort_TRIG(CLK:= Abort);
IF Execute_TRIG.Q THEN
//must see a rising edge on execute to start parsing
	starttime:= TIME();	//store the time of the beginning of execution
	parse:= TRUE;
	bufferposition:= 1;
	Done:= FALSE;
	Busy:= TRUE;
	Aborted:= FALSE;
	
	Error:= FALSE;
	ErrorPosition:= 0;
	obj_level:= 0;
	ClearNameValue();
END_IF

IF Abort_TRIG.Q THEN
	Busy:= FALSE;
	Aborted:= TRUE;
	parse:= FALSE;
END_IF

(*====================PARSE JSON STRING====================*)
//parse the input string, and start storing values in NameValue array
WHILE parse DO
	IF (JSONString^[bufferposition] = ASCII.NULL) OR (bufferposition > JSONStringSize) THEN
	//strings are terminated with a null character
	//there might not always be a null character, for example in a network buffer that is stored as an array of bytes
		parse:= FALSE;
		Done:= TRUE;
		Busy:= FALSE;
		ParseTime:= TIME() - starttime;
		RETURN;
	END_IF	
	
	CASE JSONString^[bufferposition] OF 
	ASCII.SOH..ASCII.SPACE:	// skip all control characters, including spaces
		bufferposition:= bufferposition + 1;

	ASCII.DOUBLE_QUOTE:	// " name string
		IF NameValue[obj_level].IsArray THEN
		//inside an array, look for value
			NameValue[obj_level].Value:= Value(OK=> valueok);
		ELSE
		//not an array, look for name
			NameValue[obj_level].Name:= Name(OK=> nameok);
			IF (NOT nameok) THEN
				ErrorHandler();
			END_IF	
		END_IF
				
	ASCII.OPEN_BRACE:// {, beginning of object
		OpenObject();	
		
	ASCII.CLOSE_BRACE:// }, end of object
		IF NameValue[obj_level].IsArray THEN
		//malformed string
			ErrorHandler();
		ELSE
			CloseObject();			
		END_IF
		
	ASCII.OPEN_BRACKET:	// [, beginning of array
		OpenArray();
		
	ASCII.CLOSE_BRACKET:	// ], end of array
		CloseArray();
		
	ASCII.COLON:	// :, separator for name:value pairs
		bufferposition:= bufferposition + 1;	//advance the buffer position to skip the ":"
		NameValue[obj_level].Value:= Value(OK=> valueok);	//look for value
		
	ASCII.COMMA:	// , move to next object
		Comma();
	ELSE
		IF NameValue[obj_level].IsArray THEN
		//inside an array, look for value	
			NameValue[obj_level].Value:= Value(OK=> valueok);
		ELSE
		//error, unexpected character
			ErrorHandler();			
		END_IF

	END_CASE
	
	(*========================================LOOK FOR NAMES IN LOCAL VARIABLES========================================*)
	IF valueok THEN
	//there is at least one valid name:value pair in the NameValue array--check for a match in the Config array, including nested objects
		nameok:= FALSE;
		valueok:= FALSE;
		FOR findloop:= 1 TO NumberOfVars DO
		(*loop through all configured objects and look for the name that is currently being worked on in the JSON string
		Local JSON object should be as closely matched to the expected JSON string as possible, to decrease parsing time.  
		This function will eventually find all objects, but it will start looking after the previous found variable, as it 
		is assumed that that's the most likely position for the next variable*)  
			jsonvarindex:= (jsonvarindex MOD NumberOfVars) + 1;		//increment the index of the JSONVars array
			namesmatch:= MatchAllLevels(JSONVars^[jsonvarindex]);	//check if this var matches the current object from the JSON string
			IF namesmatch THEN
				EXIT;
			END_IF
		END_FOR
	
		(*====================FOUND NAME, WRITE LOCAL VAR====================*)
		IF namesmatch THEN
		//local var name matches with JSON string name
			namesmatch:= FALSE;
			JSONVars^[jsonvarindex].AsString:= NameValue[obj_level].Value;	
		END_IF
	END_IF

	IF TIME() >= (thisloopstarttime + GPL_JSON.MAX_EXECUTION_TIME) THEN
	//this function block won't take up more than GPL_JSON.MAX_EXECUTION_TIME on one scan
	//very long strings or files could take too long to parse in one task cycle, and cause a watchdog exception
		RETURN;
	END_IF
END_WHILE

///
///| Author: Tim Van Meppelen, Pro Electric Inc.
///| timv@proelectric.com
///| Date: Oct 31, 2023
///| clear all the values in the JSONVars
METHOD ClearAll : BOOL
VAR
	i: UDINT;
END_VAR
FOR i:= 1 TO NumberOfVars DO
	JSONVars^[i].Null:= 'Null';
END_FOR
END_METHOD

///
///| Author: Tim Van Meppelen, Pro Electric Inc.
///| timv@proelectric.com
///| Date: Oct 22, 2018
///| possible value characters are any combination of the following:
///| { begin another object
///| [ begin a new array
///| " or a number or letter: value found
///| after all { and [ are found, and if any were found, the next thing will be a name string
///| loop through until a value is found, incrementing obj_level or array definitions as necessary
METHOD PRIVATE Value : STRING(GPL_JSON.MAX_VALUE_SIZE)
VAR_OUTPUT
	///a valid value was found
	OK: BOOL;
END_VAR
VAR
	lookforname: BOOL;
	///index of the beginning of a value
	value_start: UDINT;
	///index of the end of a value
	value_stop: UDINT;
	///size of value
	value_size: UDINT;
	RawValue: STRING(GPL_JSON.MAX_VALUE_SIZE);
	quotedstring: BOOL;
END_VAR
WHILE (bufferposition < JSONStringSize) DO
	
	//========== TESTS FOR SPECIAL CASES ==========
	CASE JSONString^[bufferposition] OF
		
	ASCII.SOH..ASCII.SPACE:	//skip all white space characters	
		bufferposition := bufferposition+1;
		CONTINUE;
		
	ASCII.OPEN_BRACE:// {, beginning of new object
		OpenObject();	
		lookforname:= TRUE;
		EXIT;
	
	ASCII.OPEN_BRACKET:	// [, beginning of new array
		OpenArray();
	
	ELSE
		IF lookforname THEN
		//a new object was found, and all nested objects have already been looped through, therefore this buffer position must start a new name
		//there is no value here, so exit this method, main loop in JSON_TO_STRUCT should now continue at the name, and parse its name:value pair
			RETURN;
		END_IF

		//find the beginning of the value in the buffer
		value_start:= FindValueStartPosition(QuotedString=> quotedstring);
		//find the end of the value in the buffer
		value_stop:= FindValueStopPosition(QuotedString:= quotedstring);
		//find the size of the value, and limit it to the max allowable size
		value_size:= MIN(value_stop - value_start + 1, GPL_JSON.MAX_VALUE_SIZE);
		//copy raw string into a temporary variable
		StrCpyA(
			pBuffer:= ADR(RawValue),
			iBufferSize:= UDINT_TO_DINT(value_size + 1),	//add null character
			pStr:= ADR(JSONString^[value_start])
		);			
		//validate string, and handle special characters
		Value:= JSON_TO_IEC(RawValue);
		OK:= TRUE;
		RETURN;	

	END_CASE
END_WHILE
END_METHOD

METHOD PRIVATE FindValueStartPosition : UDINT
VAR_OUTPUT
	QuotedString: BOOL;
END_VAR
VAR
	j: UDINT;
END_VAR
//========== FIND START POSITION OF VALUE ==========
FOR j:= bufferposition TO JSONStringSize DO
	CASE JSONString^[bufferposition] OF
	ASCII.DOUBLE_QUOTE:
	//value starts with a quote character
		FindValueStartPosition:= bufferposition + 1;
		bufferposition:= bufferposition + 2;
		QuotedString:= TRUE;
		RETURN;
	ELSE	
	//non-quoted, non-escaped value		
		FindValueStartPosition:= bufferposition;
		bufferposition:= bufferposition + 1;
		QuotedString:= FALSE;	
		RETURN;
	END_CASE;
END_FOR
END_METHOD

METHOD PRIVATE GetValueAsString : STRING(GPL_JSON.MAX_VALUE_SIZE)
VAR_INPUT
	RawValue: STRING(GPL_JSON.MAX_VALUE_SIZE);
END_VAR
VAR_OUTPUT
	OK: BOOL;
END_VAR
VAR
	j: UDINT;
	k: UDINT;
	pString: POINTER TO ARRAY[1..GPL_JSON.MAX_VALUE_SIZE] OF ASCII;
	temp: STRING;
END_VAR
//MOVED TO FUNCTION JSON_TO_IEC

OK:= TRUE;
pString:= ADR(RawValue);

FOR j:= 1 TO GPL_JSON.MAX_VALUE_SIZE DO
	CASE pString^[j] OF
	ASCII.NULL:
	//end of string
		RETURN;
	

	//ASCII._0:
		//IF JSONString^[j+1] = ASCII._x_ THEN
		//'0x' string, possibly indicating a hex value
		//TO DO: maybe just leave it here and deal with it in JSONVAR.AsString	
		//END_IF
		
	ASCII.BACKSLASH:
	//escape character, value starts after "\" and character
		j:= j + 1;
		CASE pString^[j] OF
		// test next position
		ASCII.DOUBLE_QUOTE:
			GetValueAsString:= CONCAT(GetValueAsString, '"');
		ASCII.BACKSLASH:
			GetValueAsString:= CONCAT(GetValueAsString, '\');	 
		ASCII.SLASH:
			GetValueAsString:= CONCAT(GetValueAsString, '/');	 
		ASCII._b_:	//backspace
			//GetValueAsString:= CONCAT(GetValueAsString, '');
			//skip this, I don't know how to implement it	 
		ASCII._f_:	//line feed
			GetValueAsString:= CONCAT(GetValueAsString, '$l');
		ASCII._n_:	//new line
			GetValueAsString:= CONCAT(GetValueAsString, '$n');	 
		ASCII._r_:	//carriage return
			GetValueAsString:= CONCAT(GetValueAsString, '$l'); 
		ASCII._t_:	//tab
			GetValueAsString:= CONCAT(GetValueAsString, '$t');
		ASCII._u_:	//unicode special character
			j:= j + 1; 		
			FOR k:= j TO j+4 DO
			//copy all characters after the escape sequence, to the end of the string
			//NOTE: this does not check for validity of hex values
				//clear previous value
				SysMemSet(
					pDest:= ADR(temp),
					udiValue:= 0,
					udiCount:= SIZEOF(temp),
				);
				//copy character into temp buffer
				SysMemCpy(
					pDest:= ADR(temp),
					pSrc:= ADR(pString^[k]),
					udiCount:= 1
				);
				//append temp buffer into output
				StrConcatA(
					pstFrom:= ADR(temp),
					pstTo:= ADR(GetValueAsString),
					iBufferSize:= SIZEOF(GetValueAsString),
				);
			END_FOR
			j:= j + 4;	
		ELSE
		//invalid escape character
			OK:= FALSE;
			RETURN;
		END_CASE;
	ELSE
	//not an escape character, copy
		//clear previous value
		SysMemSet(
			pDest:= ADR(temp),
			udiValue:= 0,
			udiCount:= SIZEOF(temp),
		);
		//copy character into temp buffer
		SysMemCpy(
			pDest:= ADR(temp),
			pSrc:= ADR(pString^[j]),
			udiCount:= 1
		);
		//append temp buffer into output
		StrConcatA(
			pstFrom:= ADR(temp),
			pstTo:= ADR(GetValueAsString),
			iBufferSize:= SIZEOF(GetValueAsString),
		);
	END_CASE
	
END_FOR
END_METHOD

METHOD PRIVATE FindValueStopPosition : UDINT
VAR_INPUT
	///value is contained within a quoted string
	QuotedString: BOOL;
END_VAR
VAR
	j: UDINT;
END_VAR
//========== FIND END POSITION OF VALUE ==========
FOR j:= bufferposition TO JSONStringSize DO
	IF JSONString^[j] = ASCII.BACKSLASH THEN
	//escape character, skip it and the next one
		j:= j + 1;
		CONTINUE;
		
	ELSIF QuotedString AND JSONString^[j] = ASCII.DOUBLE_QUOTE THEN
	//inside a quoted string, look for the next unescaped double quote
		FindValueStopPosition:= j - 1;
		bufferposition:= j + 1;	//main loop can resume at the next character after the quote
		RETURN;	
		
	ELSIF (NOT QuotedString) AND 
		(JSONString^[j] = ASCII.COMMA OR JSONString^[j] = ASCII.CLOSE_BRACE OR JSONString^[j] = ASCII.CLOSE_BRACKET) THEN
	//not in a quoted string, look for another closing character
		FindValueStopPosition:= j - 1;
		bufferposition:= j;	//rescan the character in the main loop
		RETURN;	
	
	END_IF
END_FOR
END_METHOD

///
///| Author: Tim Van Meppelen, Pro Electric Inc.
///| timv@proelectric.com
///| Date: Oct 22, 2018
///| Unexpected or invalid character found, end parsing
METHOD PRIVATE ErrorHandler
parse:= FALSE;
Busy:= FALSE;
Error:= TRUE;
ErrorMsg:= CONCAT('Unexpected character at position ', UDINT_TO_STRING(bufferposition));
ErrorPosition:= bufferposition;	//save buffer position of unexpected character
END_METHOD

METHOD PRIVATE ClearNameValue
VAR
	i: UDINT;
	j: UDINT;
END_VAR
FOR i := 1 TO GPL_JSON.MAX_LEVELS DO
    NameValue[i].Name := '';
    NameValue[i].Value := '';
    NameValue[i].IsArray := FALSE;
    NameValue[i].ArrayIndex := ARRAY_INDEX.Invalid;
    NameValue[i].ArrayDimCount := 0;
    FOR j := 1 TO GPL_JSON.MAX_ARRAY_DIMENSIONS DO
        NameValue[i].ArrayIndexes[j] := ARRAY_INDEX.Invalid;
    END_FOR
    ArrayOverflowDepth[i] := 0;
    ArrayTrackedDepth[i] := 0;
END_FOR
END_METHOD

METHOD PRIVATE CheckApplicationName : BOOL
CheckApplicationName:= TRUE;
IF (JSONVars^[1].ApplicationLevel = 0) THEN
	//maybe your application is not named 'Application'.
	//Please set proper name in library manager in GPL_JSON.APPLICATION_NAME
	Error:= TRUE;
	ErrorMsg:= 'Check application name in GPL_JSON.APPLICATION_NAME';
	CheckApplicationName:= FALSE;
END_IF
END_METHOD

METHOD PRIVATE CheckMaxVars : BOOL
CheckMaxVars:= TRUE;
IF (NumberOfVars > GPL_JSON.MAX_VARS) THEN
//need to increase GPL_JSON.MAX_VARS
	Error:= TRUE;
	ErrorMsg:= 'Too many variables, increase GPL_JSON.MAX_VARS';
	CheckMaxVars:= FALSE;
END_IF
END_METHOD

METHOD PRIVATE CheckPointers : BOOL
CheckPointers:= TRUE;
IF (JSONString = 0) OR (JSONVars = 0) THEN
//pointer invalid
	Error:= TRUE;
	ErrorMsg:= 'Input pointer invalid';
	CheckPointers:= FALSE;
END_IF
END_METHOD

///
///| Author: Tim Van Meppelen, Pro Electric Inc.
///| timv@proelectric.com
///| Date: Oct 30, 2023
///| example:  
///| {"obj1":{"obj2":{"obj3"}}}
///| NameValue array will look like this:
///| NameValue[1].Name = obj1
///| NameValue[2].Name = obj2
///| NameValue{3].Name = obj3
///| JSONVAR.Names[1] must = obj1
///| JSONVAR.Names[2] must = obj2
///| JSONVAR.Names[3] must = obj3
///
///| this method will return false on first mismatch
METHOD PRIVATE MatchAllLevels : BOOL
VAR_IN_OUT
	i_JSONVar: JSONVAR;
END_VAR
VAR
	i: UINT;
END_VAR
FOR i:= 1 TO obj_level DO
//Match name and array index.  Array index will be 0 if the current name:value is not part of an array
	IF MATCH_NAMES(i_JSONVar.JSONVarInfo[i], NameValue[obj_level-(i-1)]) THEN	
		MatchAllLevels:= TRUE;	//name in JSON string matches the local variable name
	ELSE
		MatchAllLevels:= FALSE;	//name in JSON string does not match the local variable name, go to next name
		EXIT;
	END_IF
END_FOR
END_METHOD

///
///| Author: Tim Van Meppelen, Pro Electric Inc.
///| timv@proelectric.com
///| Date: Oct 22, 2018
///| end of an object, move down in the object hierarchy
METHOD PRIVATE CloseObject
VAR
	shiftindex: INT;
END_VAR
NameValue[obj_level].Name:= '';
NameValue[obj_level].Value:= '';
NameValue[obj_level].IsArray:= FALSE;
NameValue[obj_level].ArrayIndex:= ARRAY_INDEX.Invalid;
NameValue[obj_level].ArrayDimCount:= 0;
FOR shiftindex := 1 TO TO_INT(GPL_JSON.MAX_ARRAY_DIMENSIONS) DO
    NameValue[obj_level].ArrayIndexes[shiftindex] := ARRAY_INDEX.Invalid;
END_FOR
ArrayOverflowDepth[obj_level] := 0;
ArrayTrackedDepth[obj_level] := 0;
obj_level:= obj_level - 1;
bufferposition:= bufferposition + 1;
END_METHOD

///
///| Author: Tim Van Meppelen, Pro Electric Inc.
///| timv@proelectric.com
///| Date: Oct 22, 2018
///| found the beginning of an array, set array definition at this object level
METHOD PRIVATE OpenArray
IF obj_level = 0 THEN
    obj_level := 1;
END_IF

NameValue[obj_level].IsArray := TRUE;
ArrayOverflowDepth[obj_level] := ArrayOverflowDepth[obj_level] + 1;

IF ArrayOverflowDepth[obj_level] <= GPL_JSON.MAX_ARRAY_DIMENSIONS THEN
    NameValue[obj_level].ArrayDimCount := NameValue[obj_level].ArrayDimCount + 1;
    NameValue[obj_level].ArrayIndexes[NameValue[obj_level].ArrayDimCount] := 1;
END_IF

ArrayTrackedDepth[obj_level] := NameValue[obj_level].ArrayDimCount;

IF NameValue[obj_level].ArrayDimCount = 0 THEN
    NameValue[obj_level].ArrayIndex := ARRAY_INDEX.Invalid;
ELSE
    NameValue[obj_level].ArrayIndex := NameValue[obj_level].ArrayIndexes[NameValue[obj_level].ArrayDimCount];
END_IF

bufferposition := bufferposition + 1;
END_METHOD

///
///| Author: Tim Van Meppelen, Pro Electric Inc.
///| timv@proelectric.com
///| Date: Oct 22, 2018
///| found a comma, move on to the next object	
METHOD PRIVATE Comma
IF NameValue[obj_level].IsArray THEN
    IF NameValue[obj_level].ArrayDimCount > 0 THEN
        IF ArrayOverflowDepth[obj_level] <= NameValue[obj_level].ArrayDimCount THEN
            NameValue[obj_level].ArrayIndexes[NameValue[obj_level].ArrayDimCount] :=
                NameValue[obj_level].ArrayIndexes[NameValue[obj_level].ArrayDimCount] + 1;
        ELSIF NOT GPL_JSON.FLATTEN_OVERFLOW_INTO_LAST_DIM  THEN
            NameValue[obj_level].ArrayIndexes[NameValue[obj_level].ArrayDimCount] :=
                NameValue[obj_level].ArrayIndexes[NameValue[obj_level].ArrayDimCount] + 1;
        END_IF
        NameValue[obj_level].ArrayIndex :=
            NameValue[obj_level].ArrayIndexes[NameValue[obj_level].ArrayDimCount];
    ELSE
        NameValue[obj_level].ArrayIndex := NameValue[obj_level].ArrayIndex + 1;
    END_IF
END_IF

bufferposition := bufferposition + 1;
END_METHOD

///
///| Author: Tim Van Meppelen, Pro Electric Inc.
///| timv@proelectric.com
///| Date: Oct 22, 2018
///| end of an array
METHOD PRIVATE CloseArray
IF ArrayOverflowDepth[obj_level] > 0 THEN
    IF (ArrayOverflowDepth[obj_level] <= NameValue[obj_level].ArrayDimCount)
       AND (NameValue[obj_level].ArrayDimCount > 0) THEN
        NameValue[obj_level].ArrayIndexes[NameValue[obj_level].ArrayDimCount] := ARRAY_INDEX.Invalid;
        NameValue[obj_level].ArrayDimCount := NameValue[obj_level].ArrayDimCount - 1;
    END_IF
    ArrayOverflowDepth[obj_level] := ArrayOverflowDepth[obj_level] - 1;
END_IF

ArrayTrackedDepth[obj_level] := NameValue[obj_level].ArrayDimCount;

IF ArrayOverflowDepth[obj_level] = 0 THEN
    NameValue[obj_level].IsArray := FALSE;
END_IF

IF NameValue[obj_level].ArrayDimCount = 0 THEN
    NameValue[obj_level].ArrayIndex := ARRAY_INDEX.Invalid;
ELSE
    NameValue[obj_level].ArrayIndex := NameValue[obj_level].ArrayIndexes[NameValue[obj_level].ArrayDimCount];
END_IF

bufferposition := bufferposition + 1;
END_METHOD

///
///| Author: Tim Van Meppelen, Pro Electric Inc.
///| timv@proelectric.com
///| Date: Oct 22, 2018
///| found the beginning of a new object, increment the object level
METHOD PRIVATE OpenObject
VAR
	shiftindex: INT;
END_VAR
obj_level:= obj_level + 1;	//move up a level in the object hierarchy
bufferposition:= bufferposition + 1;
END_METHOD

///
///| Author: Tim Van Meppelen, Pro Electric Inc.
///| timv@proelectric.com
///| Date: Oct 22, 2018
///| found the first quote at the beginning of a name string,
///| extract the name string and put it into the NameValue array
///| NOTE: it is technically possible in JSON to have escaped quotes in a name.  This is not possible in IEC6131
METHOD PRIVATE Name : STRING(GPL_JSON.MAX_NAME_SIZE)
VAR_OUTPUT
	///a valid name was found
	OK: BOOL;
END_VAR
VAR
	j: UDINT;
	///index of the beginning of a name
	name_start: UDINT;
	///index of the end of a name
	name_stop: UDINT;
END_VAR
name_start:= bufferposition + 1;
FOR j:= name_start TO (name_start+GPL_JSON.MAX_NAME_SIZE) DO
	IF (JSONString^[j] = ASCII.DOUBLE_QUOTE) THEN
	//find the closing quote of a name string
		name_stop:= j - 1;		//name ends at character before quote
		bufferposition:= j + 1;	//next loop can start after the quote
		OK:= TRUE;
		EXIT;
	END_IF
END_FOR

IF OK THEN
	StrCpyA(
		pBuffer:= ADR(Name),
		iBufferSize:= UDINT_TO_DINT(MIN((name_stop+2 - name_start), GPL_JSON.MAX_NAME_SIZE)),
		pStr:= ADR(JSONString^[name_start])
	);	
ELSE
	ErrorHandler();
END_IF
END_METHOD

END_FUNCTION_BLOCK

// Functions/JSON_TO_IEC
///
///| Author: Tim Van Meppelen, Pro Electric Inc.
///| timv@proelectric.com
///| Date: June 10, 2025
///| convert an JSON string to IEC, with the correct special characters
FUNCTION JSON_TO_IEC : STRING(GPL_JSON.MAX_VALUE_SIZE)
VAR_INPUT
	RawValue: STRING(GPL_JSON.MAX_VALUE_SIZE);
END_VAR
VAR
	i: DINT;
	foundindex: INT;
	searchstart: INT := 1;
END_VAR
VAR CONSTANT
	IEC_CHARS: ARRAY[1..9] OF STRING := ['$R$N', '$N', '$N', '$P', '$R', '$T', '/', '"', '\'];
	JSON_CHARS: ARRAY[1..9] OF STRING := ['\n', '\n', '\n', '\n', '\n', '\t', '\/', '\"', '\\'];
END_VAR

// Copy raw input to output
JSON_TO_IEC := RawValue;

FOR i:= 1 TO UPPER_BOUND(IEC_CHARS, 1) DO
//check for all special characters
	foundindex:= StrFindA(
		pst1:= ADR(JSON_TO_IEC),
		pst2:= ADR(JSON_CHARS[i]),
		uiSearchStart:= INT_TO_UINT(searchstart)
	);
	WHILE (foundindex > 0) DO
		StrReplaceA(
			pStInput              := ADR(JSON_TO_IEC),
			uiInputBufferSize     := SIZEOF(JSON_TO_IEC),
			pstReplaceWith        := ADR(IEC_CHARS[i]),
			iLengthInput          := LEN(JSON_TO_IEC),
			iLengthToReplace      := LEN(JSON_CHARS[i]),
			iLengthToReplaceWith  := LEN(IEC_CHARS[i]),
			iPosition             := foundindex
		);
		(* find next occurrence, starting after the just‑inserted text *)
		searchstart:= foundindex + LEN(IEC_CHARS[i]);
		foundindex:= StrFindA(
			pst1:= ADR(JSON_TO_IEC),
			pst2:= ADR(JSON_CHARS[i]),
			uiSearchStart:= INT_TO_UINT(searchstart)
		);
		IF (foundindex <= 0) THEN
		//not found, go to next
			EXIT;
		END_IF	
	
	END_WHILE
	IF (foundindex <= 0) THEN
	//not found, go to next
		CONTINUE;
	END_IF	
END_FOR

END_FUNCTION

// Functions/MATCH_NAMES
///
///| Author: Tim Van Meppelen, Pro Electric Inc.
///| timv@proelectric.com
///| Date: May 7, 2021
///| compare name in JSON string with local variable name
///| match when local variable name contains a leading underscore, if present
///| JSON allows some object names that are not valid variable names in IEC61131, for example "type", 
///| "3h", etc.  Workaround is to put an underscore at the beginning of the variable name.
///| this leading underscore can be changed or not used by modifying GPL_JSON.IGNORE_LEADING_CHAR
FUNCTION MATCH_NAMES : BOOL
VAR_INPUT
	///name:value in local value
	Name1: JSONVARINFO;
	///name:value from JSON string
	Name2: JSONNAMEVALUE;
END_VAR
VAR
	///name stripped of leading underscore, if present
	LocalVarName: STRING(GPL_JSON.MAX_NAME_SIZE);
END_VAR

IF (FIND(STR1 := Name1.Name, STR2 := GPL_JSON.IGNORE_LEADING_CHAR) = 1) THEN
    LocalVarName := DELETE(Name1.Name, 1, 1);
ELSE
    LocalVarName := Name1.Name;
END_IF

IF NOT ((Name1.Name = Name2.Name) OR (Name2.Name = LocalVarName)) THEN
    MATCH_NAMES := FALSE;
    RETURN;
END_IF

IF (Name1.ArrayDimCount = 0) AND (Name2.ArrayDimCount = 0) THEN
    IF (Name1.ArrayIndex = ARRAY_INDEX.Invalid) AND (Name2.ArrayIndex = ARRAY_INDEX.Invalid) THEN
        MATCH_NAMES := TRUE;
    ELSE
        MATCH_NAMES := (Name1.ArrayIndex = Name2.ArrayIndex);
    END_IF
    RETURN;
END_IF

IF (Name1.ArrayDimCount = 0) XOR (Name2.ArrayDimCount = 0) THEN
    MATCH_NAMES := FALSE;
    RETURN;
END_IF

MATCH_NAMES := ARRAY_INDEXES_EQUAL(
    A := Name1.ArrayIndexes,
    ACount := Name1.ArrayDimCount,
    B := Name2.ArrayIndexes,
    BCount := Name2.ArrayDimCount
);

END_FUNCTION

// Functions/ARRAY_INDEXES_EQUAL
FUNCTION ARRAY_INDEXES_EQUAL : BOOL
VAR_INPUT
	A: ARRAY[1..GPL_JSON.MAX_ARRAY_DIMENSIONS] OF INT;
	ACount: UINT;
	B: ARRAY[1..GPL_JSON.MAX_ARRAY_DIMENSIONS] OF INT;
	BCount: UINT;
END_VAR
VAR
	i: UINT;
END_VAR

IF ACount <> BCount THEN
    ARRAY_INDEXES_EQUAL := FALSE;
    RETURN;
END_IF

FOR i := 1 TO ACount DO
    IF A[i] <> B[i] THEN
        ARRAY_INDEXES_EQUAL := FALSE;
        RETURN;
    END_IF
END_FOR

ARRAY_INDEXES_EQUAL := TRUE;

END_FUNCTION

// Function Blocks/STRUCT_TO_JSON
///
///| Author: Tim Van Meppelen, Pro Electric Inc.
///| timv@proelectric.com
///| Date: Nov 2, 2018
///| Last Modified: Jan 4, 2022
///| create a JSON string from a structure of JSONVAR types
FUNCTION_BLOCK STRUCT_TO_JSON
VAR_INPUT
	///rising edge triggers compose of JSON string
	Execute: BOOL;
	///rising edge stops composing a JSON string
	Abort: BOOL;
	///pointer to JSON string
	JSONString: POINTER TO ARRAY[1..GPL_JSON.MAX_JSON_STRING] OF ASCII;
	///size of string
	JSONStringSize: DINT;
	///pointer to local structure made up of type JSONVAR
	JSONVars: POINTER TO ARRAY[1..GPL_JSON.MAX_VARS] OF JSONVAR;
	///number of variables in the local structure or array
	NumberOfVars: UDINT;
	///Suppress the codesys variable name appearing as root object (Default value is set by lib parameters)
	Rootless: BOOL := GPL_JSON.ROOTLESS;
	///don't create objects with null value
	IgnoreNull: BOOL;
	///add white space and indenting to the resulting string
	Format: BOOL;
	///max level at which to create objects
	MaxLevel: INT;
END_VAR
VAR_OUTPUT
	///busy composing a string
	Busy: BOOL;
	///successfully composed the whole string with no errors
	Done: BOOL;
	///compose aborted by Abort input
	Aborted: BOOL;
	///unexpected character detected, string not completely composed
	Error: BOOL;
	///index of local object at which composing stopped
	ErrorPosition: UDINT;
	///time it took to compose the string
	ComposeTime: TIME;
	///error information
	ErrorMsg: STRING;
END_VAR
VAR
	///current position in the string
	bufferposition: DINT;
	jsonvarindex: UDINT;
	compose: BOOL;
	///string created by current variable
	objectstr: STRING(255);
	///helper variable for names array property
	VarInfo: ARRAY[1..GPL_JSON.MAX_LEVELS] OF JSONVARINFO;
	varinfoindex: INT;
	i: UINT;
	Execute_TRIG: R_TRIG;
	Abort_TRIG: R_TRIG;
	///time the current loop started
	thisloopstarttime: TIME;
	///time composing started
	starttime: TIME;
	maxlevelindex: INT;
	objectLevel: INT;
	lastindex: UDINT;
	closeindex: UDINT;
	InitDn: BOOL;
	firstItemWritten: BOOL;
	FormatOK: BOOL;
	composethisvar: BOOL;
	///Patch
	arrayLevel: INT;
	rootLevelIndex: INT;
	offsetPrev: INT;
	offsetNext: INT;
	prevlevelindex: INT;
	nextlevelindex: INT;
	currCount: UINT;
	prevCount: UINT;
	nextCount: UINT;
	openDims: UINT;
	closeDims: UINT;
	dim: UINT;
	mustWriteArrayName:BOOL;
	samePrevArray: BOOL;
	sameNextArray: BOOL;
	currIdx: INT;
	prevIdx: INT;
	nextIdx: INT;
END_VAR

//input checks
IF NOT CheckPointers() THEN RETURN; END_IF;
IF NOT CheckMaxVars() THEN RETURN; END_IF;
IF NOT CheckApplicationName() THEN RETURN; END_IF;

thisloopstarttime:= TIME();
Execute_TRIG(CLK:= Execute);
Abort_TRIG(CLK:= Abort);

IF Execute_TRIG.Q THEN
	Initialize();
	Error:= FALSE;
	Done:= FALSE;
	Busy:= TRUE;
	Aborted:= FALSE;
	compose:= TRUE;
END_IF

IF Abort_TRIG.Q THEN
	Busy:= FALSE;
	Aborted:= TRUE;
	compose:= FALSE;
END_IF

WHILE compose AND (jsonvarindex <= lastindex) AND (bufferposition < JSONStringSize) DO
	IF (jsonvarindex = 1) THEN
		objectstr:= '{';
		firstItemWritten := FALSE;
	ELSE
		objectstr:= '';
	END_IF

	VarInfo:= JSONVars^[jsonvarindex].JSONVarInfo;
	maxlevelindex:= FindMaxLevel();

	rootLevelIndex := JSONVars^[jsonvarindex].ApplicationLevel - 2;
	IF rootLevelIndex < 1 THEN
		rootLevelIndex := 1;
	END_IF
	IF rootLevelIndex > maxlevelindex THEN
		rootLevelIndex := maxlevelindex;
	END_IF

	closeindex:= FindMatchingClose(jsonvarindex);
	composethisvar:= HasNonNullDescendant(jsonvarindex, closeindex, 2) OR (NOT IgnoreNull);

	FOR varinfoindex:= maxlevelindex TO 1 BY -1 DO
		currCount := VarInfo[varinfoindex].ArrayDimCount;
		IF (currCount = 0) AND (VarInfo[varinfoindex].ArrayIndex <> ARRAY_INDEX.Invalid) THEN
			currCount := 1;
		END_IF

		prevCount := 0;
		samePrevArray := FALSE;
		IF (jsonvarindex > 1) THEN
			offsetPrev := JSONVars^[jsonvarindex].ApplicationLevel - JSONVars^[jsonvarindex-1].ApplicationLevel;
			prevlevelindex := varinfoindex - offsetPrev;
			IF (prevlevelindex >= 1) AND (prevlevelindex <= GPL_JSON.MAX_LEVELS) THEN
				prevCount := JSONVars^[jsonvarindex-1].JSONVarInfo[prevlevelindex].ArrayDimCount;
				IF (prevCount = 0) AND (JSONVars^[jsonvarindex-1].JSONVarInfo[prevlevelindex].ArrayIndex <> ARRAY_INDEX.Invalid) THEN
					prevCount := 1;
				END_IF

				IF (prevCount > 0)
					AND (JSONVars^[jsonvarindex-1].JSONVarInfo[prevlevelindex].Name = VarInfo[varinfoindex].Name) THEN
					samePrevArray := TRUE;
				END_IF
			END_IF
		END_IF

		openDims := 0;
		IF (currCount > 0) THEN
			IF NOT samePrevArray THEN
				openDims := currCount;
			ELSE
				FOR dim := 1 TO currCount DO
					IF (dim <= VarInfo[varinfoindex].ArrayDimCount) THEN
						currIdx := VarInfo[varinfoindex].ArrayIndexes[dim];
					ELSE
						currIdx := VarInfo[varinfoindex].ArrayIndex;
					END_IF

					IF (dim <= JSONVars^[jsonvarindex-1].JSONVarInfo[prevlevelindex].ArrayDimCount) THEN
						prevIdx := JSONVars^[jsonvarindex-1].JSONVarInfo[prevlevelindex].ArrayIndexes[dim];
					ELSE
						prevIdx := JSONVars^[jsonvarindex-1].JSONVarInfo[prevlevelindex].ArrayIndex;
					END_IF

					IF (currIdx < prevIdx) THEN
						openDims := openDims + 1;
					END_IF
				END_FOR
			END_IF
		END_IF
		
		IF (openDims > 0)
		  AND composethisvar
		  AND NOT (Rootless AND (varinfoindex = rootLevelIndex)) THEN
			PrependComma();
			mustWriteArrayName := NOT samePrevArray;
			IF samePrevArray
			   AND (jsonvarindex > 1)
			   AND (prevlevelindex >= 1)
			   AND (prevlevelindex <= GPL_JSON.MAX_LEVELS)
			   AND JSONVars^[jsonvarindex-1].JSONVarInfo[prevlevelindex].EndObject THEN
				mustWriteArrayName := TRUE;
			END_IF
			IF mustWriteArrayName THEN
				CreateName(Name:= VarInfo[varinfoindex].Name);
			END_IF
			FOR dim := 1 TO openDims DO
				CreateArray();
			END_FOR
		END_IF

		IF VarInfo[varinfoindex].NewObject AND (varinfoindex <> 1)
		 AND composethisvar
		 AND NOT (Rootless AND (varinfoindex = rootLevelIndex)) THEN
			PrependComma();
			IF (currCount = 0) THEN
				CreateName(Name:= VarInfo[varinfoindex].Name);
			END_IF
			CreateObject();
		END_IF

		IF (varinfoindex=1) THEN
			IF (VarInfo[varinfoindex].InArray
			 OR (VarInfo[varinfoindex].ArrayDimCount > 0)
			 OR (VarInfo[varinfoindex].ArrayIndex <> ARRAY_INDEX.Invalid)) THEN
				IF NOT (IgnoreNull AND (VarInfo[1].InArray) AND (JSONVars^[jsonvarindex].ValueType = JSONVALUETYPE.json_null)) THEN
					PrependComma();
					CreateValue();
				END_IF
			ELSE
				IF NOT (IgnoreNull AND (JSONVars^[jsonvarindex].ValueType = JSONVALUETYPE.json_null)) THEN
					PrependComma();
					CreateName(Name:= VarInfo[varinfoindex].Name);
					CreateValue();
				END_IF
			END_IF
		END_IF
	END_FOR

	FOR varinfoindex:= 1 TO maxlevelindex DO
		currCount := VarInfo[varinfoindex].ArrayDimCount;
		IF (currCount = 0) AND (VarInfo[varinfoindex].ArrayIndex <> ARRAY_INDEX.Invalid) THEN
			currCount := 1;
		END_IF

		nextCount := 0;
		sameNextArray := FALSE;
		IF (jsonvarindex < lastindex) THEN
			offsetNext := JSONVars^[jsonvarindex+1].ApplicationLevel - JSONVars^[jsonvarindex].ApplicationLevel;
			nextlevelindex := varinfoindex + offsetNext;
			IF (nextlevelindex >= 1) AND (nextlevelindex <= GPL_JSON.MAX_LEVELS) THEN
				nextCount := JSONVars^[jsonvarindex+1].JSONVarInfo[nextlevelindex].ArrayDimCount;
				IF (nextCount = 0) AND (JSONVars^[jsonvarindex+1].JSONVarInfo[nextlevelindex].ArrayIndex <> ARRAY_INDEX.Invalid) THEN
					nextCount := 1;
				END_IF

				IF (nextCount > 0)
					AND (JSONVars^[jsonvarindex+1].JSONVarInfo[nextlevelindex].Name = VarInfo[varinfoindex].Name) THEN
					sameNextArray := TRUE;
				END_IF
			END_IF
		END_IF

		closeDims := 0;
		IF (currCount > 0) THEN
			IF NOT sameNextArray THEN
				closeDims := currCount;
			ELSE
				FOR dim := 1 TO currCount DO
					IF (dim <= JSONVars^[jsonvarindex+1].JSONVarInfo[nextlevelindex].ArrayDimCount) THEN
						nextIdx := JSONVars^[jsonvarindex+1].JSONVarInfo[nextlevelindex].ArrayIndexes[dim];
					ELSE
						nextIdx := JSONVars^[jsonvarindex+1].JSONVarInfo[nextlevelindex].ArrayIndex;
					END_IF

					IF (dim <= VarInfo[varinfoindex].ArrayDimCount) THEN
						currIdx := VarInfo[varinfoindex].ArrayIndexes[dim];
					ELSE
						currIdx := VarInfo[varinfoindex].ArrayIndex;
					END_IF

					IF (nextIdx < currIdx) THEN
						closeDims := closeDims + 1;
					END_IF
				END_FOR
			END_IF
		END_IF

		IF (varinfoindex <> 1) AND VarInfo[varinfoindex].EndObject
			AND NOT (Rootless AND (varinfoindex = rootLevelIndex)) THEN
			CloseObject();
		END_IF

		IF (closeDims > 0)
			AND NOT (Rootless AND (varinfoindex = rootLevelIndex)) THEN
			FOR dim := 1 TO closeDims DO
				CloseArray();
			END_FOR
		END_IF
	END_FOR

	StrConcatA(
		pstFrom:= ADR(objectstr),
		pstTo:= ADR(JSONString^[bufferposition]),
		iBufferSize:= DINT_TO_INT(JSONStringSize)
	);
	bufferposition:= bufferposition + LEN(objectstr);

	IF (bufferposition >= JSONStringSize) THEN
		Busy:= FALSE;
		Done:= FALSE;
		Error:= TRUE;
		ErrorMsg:= 'JSONString too small';
		compose:= FALSE;
	END_IF

	IF (jsonvarindex >= NumberOfVars) THEN
		compose:= FALSE;
		Busy:= FALSE;
		Done:= TRUE;
		ComposeTime:= TIME() - starttime;
		JSONString^[bufferposition]:= ASCII.CLOSE_BRACE;
		bufferposition:= bufferposition + 1;
		JSONString^[bufferposition]:= ASCII.NULL;

		IF Format THEN
			FormatOK:= FORMAT_JSON(JSONString, JSONStringSize);
			IF (NOT FormatOK) THEN
				Error:= TRUE;
				ErrorMsg:= 'Formatting failed, check string size';
			END_IF
		END_IF
	ELSE
		jsonvarindex:= jsonvarindex + 1;
	END_IF

	IF TIME() >= (thisloopstarttime + GPL_JSON.MAX_EXECUTION_TIME) THEN
		RETURN;
	END_IF
END_WHILE

///
///| Author: Tim Van Meppelen, Pro Electric Inc.
///| timv@proelectric.com
///| Date: June 5, 2025
///| determine the highest level to compose to
METHOD PRIVATE FindMaxLevel : INT
IF (MaxLevel = 0) THEN
//default, create all objects below the program level
	FindMaxLevel:= JSONVars^[jsonvarindex].ApplicationLevel - 2;
ELSE
//manually defined with the MaxLevel input
	FindMaxLevel:= MaxLevel;
END_IF
END_METHOD

///
///| Author: Tim Van Meppelen, Pro Electric Inc.
///| timv@proelectric.com
///| Date: Oct 22, 2018
///| create a new JSON array
///| 
///| [ ------ ------------ value ---------------- ] 
///|         /                               \
///| 	      \_______________ , _____________/
///| 		
METHOD PRIVATE CreateArray
objectstr:= CONCAT(objectstr, '[');	//opening [
arrayLevel := arrayLevel + 1;  //Patch
firstItemWritten:= FALSE;
//ArrOpened[varinfoindex] := TRUE; // mark that a '[' is pending a ']'
END_METHOD

///
///| Author: Tim Van Meppelen, Pro Electric Inc.
///| timv@proelectric.com
///| Date: Oct 22, 2018
///| create a new JSON object
///| 
///| {------ "name" ------ : ----- value --------- }
///|     /                                 \
///| 	  \_______________ , _______________/
///| 
METHOD PRIVATE CreateObject
objectstr:= CONCAT(objectstr, '{');	//opening {
objectLevel := objectLevel + 1;
firstItemWritten:= FALSE;
END_METHOD

///
///| Author: Tim Van Meppelen, Pro Electric Inc.
///| timv@proelectric.com
///| Date: Oct 22, 2018
///| create a JSON value string from a local variable of type JSONVAR
METHOD PRIVATE CreateValue
CASE JSONVars^[jsonvarindex].ValueType OF
//append value to object string
JSONVALUETYPE.json_number:
	objectstr:= CONCAT(objectstr, JSONVars^[jsonvarindex].AsString);
JSONVALUETYPE.json_integer,
JSONVALUETYPE.json_uinteger:
	CASE JSONVars^[jsonvarindex].Format OF
	JSONFORMAT.Hex:
	//format number as hex
		IF GPL_JSON.JSON5 THEN
		//JSON5 hex value
			objectstr:= CONCAT(objectstr, JSONVars^[jsonvarindex].AsHexString);
		ELSE
		//JSON compliant quoted hex string 
			objectstr:= CONCAT(objectstr, '"');	//opening quote
			objectstr:= CONCAT(objectstr, JSONVars^[jsonvarindex].AsHexString);
			objectstr:= CONCAT(objectstr, '"');	//closing quote			
		END_IF
	JSONFORMAT.Unicode:
	//format number as unicode string
		objectstr:= CONCAT(objectstr, '"');	//opening quote
		objectstr:= CONCAT(objectstr, JSONVars^[jsonvarindex].AsUnicode);
		objectstr:= CONCAT(objectstr, '"');	//closing quote
	ELSE	
	//numeric value
		objectstr:= CONCAT(objectstr, JSONVars^[jsonvarindex].AsString);
	END_CASE
JSONVALUETYPE.json_boolean:
	objectstr:= CONCAT(objectstr, JSONVars^[jsonvarindex].AsString);
JSONVALUETYPE.json_string:
	objectstr:= CONCAT(objectstr, '"');	//opening quote
	objectstr:= CONCAT(objectstr, IEC_TO_JSON(JSONVars^[jsonvarindex].AsString));
	objectstr:= CONCAT(objectstr, '"');	//closing quote
JSONVALUETYPE.json_null:
	objectstr:= CONCAT(objectstr, 'null');
END_CASE
END_METHOD

///
///| Author: Tim Van Meppelen, Pro Electric Inc.
///| timv@proelectric.com
///| Date: Oct 22, 2018
///| create a JSON name string from a local variable of type JSONVAR
METHOD PRIVATE CreateName
VAR_INPUT
	Name: STRING(GPL_JSON.MAX_NAME_SIZE);
END_VAR
VAR
	indent: INT;
	leadingpos: INT;
END_VAR
objectstr:= CONCAT(objectstr, '"');	//opening quote

leadingpos:= FIND(Name, GPL_JSON.IGNORE_LEADING_CHAR);
//if leading character is configured and present, delete it from the name
IF (leadingpos = 1) THEN
	objectstr:= CONCAT(objectstr, DELETE(Name, 1, 1));//variable name
ELSE
	objectstr:= CONCAT(objectstr, Name);//variable name
END_IF

objectstr:= CONCAT(objectstr, '":');	//closing quote and name:value separator
END_METHOD

///
///| Author: Tim Van Meppelen, Pro Electric Inc.
///| timv@proelectric.com
///| Date: June 5, 2025
///| check an object or array to see if it has non-null descendents
METHOD PRIVATE HasNonNullDescendant : BOOL
VAR_INPUT
	/// current jsonvarindex
	startIndex: UDINT;
	/// closing jsonvarindex of this object
	endIndex: UDINT;
	/// namesindex we are about to open
	varinfoindex: INT;
END_VAR
VAR
	depth: INT := 0;
	i: UDINT;
	/// temp
	VarInfo: ARRAY[1..GPL_JSON.MAX_LEVELS] OF JSONVARINFO;
END_VAR
FOR i:= startIndex TO endIndex DO
	IF (JSONVars^[i].ValueType <> JSONVALUETYPE.json_null) THEN
		HasNonNullDescendant:= TRUE;
		RETURN;
	END_IF
END_FOR


// scan ahead until we close the object/array that begins at startIndex,level
FOR i := startIndex TO lastindex DO
    VarInfo := JSONVars^[i].JSONVarInfo;

    //walk matching depth so we know when the structure ends
    IF VarInfo[varinfoindex].EndObject OR VarInfo[varinfoindex].EndArray THEN
        IF depth = 0 THEN
            EXIT;                  // reached our matching close
        ELSE
            depth := depth - 1;    // coming out of nested child
        END_IF

    ELSIF VarInfo[varinfoindex].NewObject OR VarInfo[varinfoindex].NewArray THEN
        depth := depth + 1;        // going one level deeper
    END_IF

    //if the var would actually be emitted, we are done
    IF NOT (IgnoreNull AND (JSONVars^[i].ValueType = JSONVALUETYPE.json_null)) THEN
        HasNonNullDescendant := TRUE;
        RETURN;
    END_IF
END_FOR

HasNonNullDescendant := FALSE;
END_METHOD

///
///| Author: Tim Van Meppelen, Pro Electric Inc.
///| timv@proelectric.com
///| Date: June 5, 2025
///| prepend a comma if necessary
METHOD PRIVATE PrependComma : BOOL
IF NOT firstItemWritten THEN
  // do not prepend comma on very first element
  firstItemWritten := TRUE;
ELSE
  // prepend comma on all subsequent elements
  objectstr := CONCAT(objectstr, ',');
END_IF
END_METHOD

///
///| Author: Tim Van Meppelen, Pro Electric Inc.
///| timv@proelectric.com
///| Date: June 5, 2025
///| initialize variables
METHOD PRIVATE Initialize : BOOL
starttime:= TIME();
lastindex:= MIN(NumberOfVars, GPL_JSON.MAX_VARS);
IF NOT JSONVars^[1].Init THEN
	JSONVars^[1].Init := InitJsonVars();
END_IF
ErrorPosition:= 0;
bufferposition:= 1;
jsonvarindex:= 1;
objectLevel := 0;
arrayLevel := 0;

firstItemWritten := FALSE;
FOR i:= 1 TO GPL_JSON.MAX_LEVELS DO
	VarInfo[i].Name:= '';
	VarInfo[i].ArrayIndex:= ARRAY_INDEX.Invalid;
	VarInfo[i].ArrayDimCount:= 0;
END_FOR
SysMemSet(
	pDest:= JSONString,
	udiValue:= 0,
	udiCount:= DINT_TO_UDINT(JSONStringSize)
);
END_METHOD

///
///| Author: Tim Van Meppelen, Pro Electric Inc.
///| timv@proelectric.com
///| Date: June 5, 2025
///| initialize some properties of JSONVARs that can't be determined in the JSONVAR.FB_Init method
///| see note in JSONVAR.FB_Init
METHOD PRIVATE InitJsonVars : BOOL
VAR
	varlevelindex: INT;
	jsonvarindex: INT;
END_VAR
FOR varlevelindex:= 1 TO JSONVars^[1].ApplicationLevel-2 DO
	IF (JSONVars^[1].JSONVarInfo[varlevelindex].ArrayDimCount > 0)
	   OR (JSONVars^[1].JSONVarInfo[varlevelindex].ArrayIndex <> ARRAY_INDEX.Invalid) THEN
		JSONVars^[1].JSONVarInfo[varlevelindex].NewArray:= TRUE;
		IF (varlevelindex > 1) THEN
			JSONVars^[1].JSONVarInfo[varlevelindex].NewObject:= TRUE;
		END_IF
	ELSIF (varlevelindex > 1) OR (NumberofVars = 1) THEN
		JSONVars^[1].JSONVarInfo[varlevelindex].NewObject:= TRUE;
	END_IF
END_FOR

JSONVars^[1].LastIndex := lastindex;
FOR varlevelindex:= 1 TO JSONVars^[lastindex].ApplicationLevel-2 DO
	IF (JSONVars^[lastindex].JSONVarInfo[varlevelindex].ArrayDimCount > 0)
	   OR (JSONVars^[lastindex].JSONVarInfo[varlevelindex].ArrayIndex <> ARRAY_INDEX.Invalid) THEN
		JSONVars^[lastindex].JSONVarInfo[varlevelindex].EndArray:= TRUE;
		IF (varlevelindex > 1) THEN
			JSONVars^[lastindex].JSONVarInfo[varlevelindex].EndObject:= TRUE;
		END_IF
	ELSIF (varlevelindex > 1) OR (NumberofVars = 1) THEN
		JSONVars^[lastindex].JSONVarInfo[varlevelindex].EndObject:= TRUE;
	END_IF
END_FOR

InitJsonVars:= TRUE;
END_METHOD

METHOD PRIVATE CheckMaxVars : BOOL
CheckMaxVars:= TRUE;
IF (NumberOfVars > GPL_JSON.MAX_VARS) THEN
//need to increase GPL_JSON.MAX_VARS
	Error:= TRUE;
	ErrorMsg:= 'Too many variables, increase GPL_JSON.MAX_VARS';
	CheckMaxVars:= FALSE;
END_IF
END_METHOD

METHOD PRIVATE CheckApplicationName : BOOL
CheckApplicationName:= TRUE;
IF (JSONVars^[1].ApplicationLevel = 0) THEN
	//maybe your application is not named 'Application'.
	//Please set proper name in library manager in GPL_JSON.APPLICATION_NAME
	Error:= TRUE;
	ErrorMsg:= 'Check application name in GPL_JSON.APPLICATION_NAME';
	CheckApplicationName:= FALSE;
END_IF
END_METHOD

METHOD PRIVATE CheckPointers : BOOL
CheckPointers:= TRUE;
IF (JSONString = 0) OR (JSONVars = 0) THEN
//pointer invalid
	Error:= TRUE;
	ErrorMsg:= 'Input pointer invalid';
	CheckPointers:= FALSE;
END_IF
END_METHOD

///
///| Author: Tim Van Meppelen, Pro Electric Inc.
///| timv@proelectric.com
///| Date: June 5, 2025
///| find the matching close object for this level
METHOD PRIVATE FindMatchingClose : UDINT
VAR_INPUT
	/// current jsonvarindex
	startIndex: UDINT;
END_VAR
VAR
	i: UDINT;
	j: UDINT;
	newobjlevel: UDINT;
	/// temp
	VarInfoTest: ARRAY[1..GPL_JSON.MAX_LEVELS] OF JSONVARINFO;
END_VAR
FOR i:= startindex TO lastindex DO
	VarInfoTest:= JSONVars^[i].JSONVarInfo;	//helper variable
	FOR j:= 1 TO GPL_JSON.MAX_LEVELS DO
		IF VarInfo[j].NewObject THEN
		//find the level at which a new object is created
			newobjlevel:= j;
			EXIT;
		END_IF
	END_FOR
	IF newobjlevel = 0 THEN
	//this object doesn't start a new level
		FindMatchingClose:= lastindex;
		RETURN;
	END_IF
	IF VarInfoTest[newobjlevel].EndObject THEN
	//found the end object of this level
		FindMatchingClose:= i;
		RETURN;
	END_IF
END_FOR
END_METHOD

///
///| Author: Tim Van Meppelen, Pro Electric Inc.
///| timv@proelectric.com
///| Date: Oct 22, 2018
///| close a JSON array
METHOD PRIVATE CloseArray

// objectstr:= CONCAT(objectstr, ']');  //Patch
IF arrayLevel > 0 THEN //Patch
	objectstr:= CONCAT(objectstr, ']'); //Patch
	arrayLevel := arrayLevel - 1; //Patch
END_IF //Patch
END_METHOD

///
///| Author: Tim Van Meppelen, Pro Electric Inc.
///| timv@proelectric.com
///| Date: Oct 22, 2018
///| close a JSON object
METHOD PRIVATE CloseObject
VAR
	indent: INT;
END_VAR
IF objectLevel > 0 THEN
	objectstr:= CONCAT(objectstr, '}');
	objectLevel := objectLevel - 1;
END_IF
END_METHOD

///
///| Author: Tim Van Meppelen, Pro Electric Inc.
///| timv@proelectric.com
///| Oct 31, 2023
///| clear output string
METHOD ClearString : BOOL
JSONString^[1]:= ASCII.NULL;
END_METHOD

END_FUNCTION_BLOCK

// Functions/FORMAT_JSON
///
///| Author: Tim Van Meppelen, Pro Electric Inc.
///| timv@proelectric.com
///| Date: June 6, 2025
///| format a JSON string
FUNCTION FORMAT_JSON : BOOL
VAR_INPUT
	/// Pointer to the raw (unformatted) JSON
	JSONString: POINTER TO STRING(GPL_JSON.MAX_JSON_STRING);
	///SIZEOF of JSONString
	JSONSize: DINT;
END_VAR
VAR
	i: DINT;
	j: DINT;
	currentChar: ASCII;
	prevChar: ASCII;
	charAsString: STRING(1);
	indentLvl: INT;
	Buffer: STRING;
	TempString: STRING(GPL_JSON.MAX_JSON_STRING);
	inString: BOOL;
END_VAR
VAR CONSTANT
	COLON: STRING(2) := ': ';
END_VAR

FOR i := 0 TO JSONSize-1 DO
//iterate through each character
	Buffer:= '';
	currentChar:= JSONString^[i];	//convert to ASCII enumeration for CASE statement
	SysMemCpy(
		pDest:= ADR(charAsString), 
		pSrc:= ADR(JSONString^[i]), 
		udiCount:= 1
	);	//copy single string for concatenation
	
	IF (currentChar = ASCII.DOUBLE_QUOTE) AND (prevChar <> ASCII.BACKSLASH) THEN
        inString := NOT inString;
    END_IF
	prevChar:= currentChar;
	
	IF inString THEN
    //inside a string, copy characters and skip the rest of the CASE statement
		Buffer:= CONCAT(Buffer, charAsString);	
		StrConcatA(
			pstFrom:= ADR(Buffer),
			pstTo:= ADR(TempString), 
			iBufferSize:= DINT_TO_INT(JSONSize)
		);
		CONTINUE;	//skip the CASE statement
    END_IF
	
	CASE currentChar OF

	ASCII.NULL: 
	// Null character, end of string		
		EXIT;

	ASCII.OPEN_BRACE,
	ASCII.OPEN_BRACKET:
	// “{” or “[” : append it, newline, increase indent, then indent	
		Buffer:= CONCAT(Buffer, charAsString);	
		Buffer:= CONCAT(Buffer, GPL_JSON.NEWLINE);	
		indentLvl:= indentLvl + 1;
		FOR j:= 1 TO indentLvl DO
			Buffer:= CONCAT(Buffer, GPL_JSON.INDENT);
		END_FOR

	ASCII.CLOSE_BRACE,
	ASCII.CLOSE_BRACKET:
	// “}” or “]” : newline, decrease indent, indent, then append	
		Buffer:= CONCAT(Buffer, GPL_JSON.NEWLINE);		
		indentLvl:= indentLvl - 1;	
		FOR j:= 1 TO indentLvl DO
			Buffer:= CONCAT(Buffer, GPL_JSON.INDENT);
		END_FOR
		Buffer:= CONCAT(Buffer, charAsString);	

	ASCII.COMMA:
	// "," : write comma, newline, indent	
		Buffer:= CONCAT(Buffer, charAsString);				
		Buffer:= CONCAT(Buffer, GPL_JSON.NEWLINE);	
		FOR j:= 1 TO indentLvl DO
			Buffer:= CONCAT(Buffer, GPL_JSON.INDENT);
		END_FOR

	ASCII.COLON:
	// “:” : append colon and a space
		Buffer:= CONCAT(Buffer, COLON);	

	ELSE
	//any other character, append		
		Buffer:= CONCAT(Buffer, charAsString);	
	
	END_CASE;
	StrConcatA(
		pstFrom:= ADR(Buffer),
		pstTo:= ADR(TempString), 
		iBufferSize:= DINT_TO_INT(JSONSize)
	);
	
END_FOR

SysMemSet(
	pDest:= JSONString, 
	udiValue:= 0, 
	udiCount:= DINT_TO_UDINT(JSONSize)
);	//clear unformatted string

SysMemCpy(
	pDest:= JSONString, 
	pSrc:= ADR(TempString), 
	udiCount:= DINT_TO_UDINT(JSONSize)
);	//overwrite unformatted string

FORMAT_JSON := TRUE;

END_FUNCTION

// Functions/IEC_TO_JSON
///
///| Author: Tim Van Meppelen, Pro Electric Inc.
///| timv@proelectric.com
///| Date: June 10, 2025
///| convert an IEC string to JSON, with the correct escape characters
FUNCTION IEC_TO_JSON : STRING(GPL_JSON.MAX_VALUE_SIZE)
VAR_INPUT
	RawValue: STRING(GPL_JSON.MAX_VALUE_SIZE);
END_VAR
VAR
	i: DINT;
	foundindex: INT;
	searchstart: INT := 1;
END_VAR
VAR CONSTANT
	IEC_CHARS: ARRAY[1..9] OF STRING := ['$R$N', '$N', '$N', '$P', '$R', '$T', '/', '"', '\'];
	JSON_CHARS: ARRAY[1..9] OF STRING := ['\n', '\n', '\n', '\n', '\n', '\t', '\/', '\"', '\\'];
END_VAR

// Copy raw input to output
IEC_TO_JSON := RawValue;

FOR i:= 1 TO UPPER_BOUND(IEC_CHARS, 1) DO
//check for all special characters
	foundindex:= StrFindA(
		pst1:= ADR(IEC_TO_JSON),
		pst2:= ADR(IEC_CHARS[i]),
		uiSearchStart:= INT_TO_UINT(searchstart)
	);
	WHILE (foundindex > 0) DO
		StrReplaceA(
			pStInput              := ADR(IEC_TO_JSON),
			uiInputBufferSize     := SIZEOF(IEC_TO_JSON),
			pstReplaceWith        := ADR(JSON_CHARS[i]),
			iLengthInput          := LEN(IEC_TO_JSON),
			iLengthToReplace      := LEN(IEC_CHARS[i]),
			iLengthToReplaceWith  := LEN(JSON_CHARS[i]),
			iPosition             := foundindex
		);
		(* find next occurrence, starting after the just‑inserted text *)
		searchstart:= foundindex + LEN(JSON_CHARS[i]);
		foundindex:= StrFindA(
			pst1:= ADR(IEC_TO_JSON),
			pst2:= ADR(IEC_CHARS[i]),
			uiSearchStart:= INT_TO_UINT(searchstart)
		);
		IF (foundindex <= 0) THEN
		//not found, go to next
			EXIT;
		END_IF	
	
	END_WHILE
	IF (foundindex <= 0) THEN
	//not found, go to next
		CONTINUE;
	END_IF	
END_FOR

END_FUNCTION

// Functions/SPLIT_VARNAME
///
///| Author: Tim Van Meppelen, Pro Electric Inc.
///| timv@proelectric.com
///| Date: June 26, 2018
///| split a string into an array at the '.' character
///| modified from https://forum.codesys.com/viewtopic.php?t=9889
///| 'a.b.c.d' becomes an array[1]=d, [2]=c, [3]=b, [4]=a
FUNCTION SPLIT_VARNAME : UINT
VAR_INPUT
	VarNameArray: REFERENCE TO ARRAY [1..GPL_JSON.MAX_LEVELS] OF JSONVARINFO;
	///input string
	StringIn: STRING(GPL_JSON.MAX_VAR_NAME);
END_VAR
VAR CONSTANT
	SPLIT_CHAR: STRING(1) := '.';
END_VAR
VAR
	ArraySize: UINT := 1;
	sShortString: STRING;
	iSplitLocation: INT;
	i: UINT;
	TempArray: ARRAY[1..GPL_JSON.MAX_LEVELS] OF STRING;
END_VAR

//Loop through string until there is no string left or array has hit its limits
WHILE (StrLenA(pstData:= ADR(StringIn)) > 0) DO
	//Find location of first break point
	iSplitLocation := StrFindA(
		pst1:= ADR(StringIn), 
		pst2:= ADR(SPLIT_CHAR), 
		uiSearchStart:= 1
	) - 1;
	
	//If there is no break point found then set location to size of string
	IF (iSplitLocation = -1) THEN
		iSplitLocation := DINT_TO_INT(StrLenA(pstData:= ADR(StringIn)));
	END_IF
  
	//Copy the part of the string that is needed for the parameter.
	StrMidA(
		pst:= ADR(StringIn), 
		uiInputBufferSize:= SIZEOF(StringIn), 
		iLength:= iSplitLocation, 
		iPosition:= 1, 
		pstResult:= ADR(sShortString), 
		uiResultBufferSize:= SIZEOF(sShortString)
	);

	//Make sure string is not empty before using up an array spot.
	IF (StrLenA(pstData:= ADR(sShortString)) > 0) THEN
		TempArray[ArraySize] := sShortString;
		ArraySize := ArraySize + 1;
	END_IF

	//Remove copied components from long string
	StrDeleteA(
		pby:= ADR(StringIn), 
		iLength:= (iSplitLocation + LEN(SPLIT_CHAR)), 
		iPosition:= 1
	);

	//Check to see if more parameters can fit in array. If not exit loop
	IF (ArraySize > GPL_JSON.MAX_LEVELS) THEN
		EXIT;
	END_IF 
END_WHILE

ArraySize:= ArraySize - 1;

FOR i:= 0 TO ArraySize-1 DO
//reverse the order of the array
	VarNameArray[i+1].Name:= TempArray[ArraySize-i];	
END_FOR

SPLIT_VARNAME:= ArraySize;

END_FUNCTION

// Functions/HEXSTR_TO_UDINT
///
///| Description:
///| This function converts a string representing a hexadecimal number
///| into a UDINT (Unsigned Double Integer) value.
///| The string may optionally start with '0x' or '0X'.
///| 
///| Example inputs: 'FF' -> 255, '0xFF' -> 255, '1A3' -> 419, '0x12345678' -> 305419896
///| 
///| Limitations:
///| - The maximum length of the hexadecimal string (excluding '0x') is 8 characters,
///|   since a UDINT is a 32-bit integer (2^32 - 1), which corresponds to FFFFFFFF in hexadecimal.
///| 
///| Author: Fabrizio Morlino
///| Date: 20/05/2025
FUNCTION HEXSTR_TO_UDINT : UDINT
VAR_INPUT
	/// Hex string to convert 
	sHex: STRING;
END_VAR
VAR_OUTPUT
	xError: BOOL;
END_VAR
VAR
	/// Index for iteration
	i: INT;
	/// Current character
	c: BYTE;
	/// Numeric value of the hexadecimal character
	digit: BYTE;
	/// Final result
	result: UDINT := 0;
	/// Length of the string
	sHexLen: INT;
	/// Start index after the prefix
	startIdx: INT := 0;
END_VAR

// Removes the '0x' or '0X' prefix if present
IF (LEFT(sHex, 2) = '0x') OR (LEFT(sHex, 2) = '0X') THEN
    startIdx := 2;
END_IF;

sHexLen := LEN(sHex);

// If the string is empty after the prefix
IF sHexLen - startIdx <= 0 THEN
	xError := TRUE;
	RETURN;
END_IF

// If the hexadecimal string is too large for a UDINT
IF sHexLen - startIdx > 8 THEN
	xError := TRUE;
	RETURN;
END_IF

